LIN {X 0,Y 495.038,Z 903.66,A -85,B 0,C 180,E1 20472.506,E2 20472.506} C_VEL
LIN {X 0,Y 497.453,Z 905.615,A -85,B 0,C 180,E1 20472.244,E2 20472.244} C_VEL
LIN {X 0,Y 483.412,Z 928.293,A -85,B 0,C 180,E1 20471.672,E2 20471.672} C_VEL
LIN {X 0,Y 473.515,Z 947.117,A -85,B 0,C 180,E1 20471.077,E2 20471.077} C_VEL
LIN {X 0,Y 466.181,Z 963.721,A -85,B 0,C 180,E1 20470.451,E2 20470.451} C_VEL
LIN {X 0,Y 458.344,Z 980.789,A -85,B 0,C 180,E1 20469.812,E2 20469.812} C_VEL
LIN {X 0,Y 450.078,Z 1004.055,A -85,B 0,C 180,E1 20468.798,E2 20468.798} C_VEL
LIN {X 0,Y 447.354,Z 1025.742,A -85,B 0,C 180,E1 20468.553,E2 20468.553} C_VEL
LIN {X 0,Y 446.305,Z 1053.945,A -85,B 0,C 180,E1 20467.96,E2 20467.96} C_VEL
LIN {X 0,Y 444.603,Z 1079.758,A -85,B 0,C 180,E1 20467.185,E2 20467.185} C_VEL
LIN {X 0,Y 442.821,Z 1103.831,A -85,B 0,C 180,E1 20466.222,E2 20466.222} C_VEL
LIN {X 0,Y 440.838,Z 1127.571,A -85,B 0,C 180,E1 20465.018,E2 20465.018} C_VEL
LIN {X 0,Y 438.693,Z 1150.972,A -85,B 0,C 180,E1 20463.553,E2 20463.553} C_VEL
LIN {X 0,Y 436.639,Z 1172.47,A -85,B 0,C 180,E1 20461.936,E2 20461.936} C_VEL
LIN {X 0,Y 434.521,Z 1192.931,A -85,B 0,C 180,E1 20460.108,E2 20460.108} C_VEL
LIN {X 0,Y 432.447,Z 1212.213,A -85,B 0,C 180,E1 20458.068,E2 20458.068} C_VEL
LIN {X 0,Y 430.487,Z 1230.142,A -85,B 0,C 180,E1 20455.817,E2 20455.817} C_VEL
LIN {X 0,Y 428.709,Z 1246.625,A -85,B 0,C 180,E1 20453.359,E2 20453.359} C_VEL
LIN {X 0,Y 427.372,Z 1259.283,A -85,B 0,C 180,E1 20451.119,E2 20451.119} C_VEL
LIN {X 0,Y 426.348,Z 1269.529,A -85,B 0,C 180,E1 20449.025,E2 20449.025} C_VEL
LIN {X 0,Y 425.398,Z 1280.533,A -85,B 0,C 180,E1 20446.383,E2 20446.383} C_VEL
LIN {X 0,Y 424.715,Z 1289.348,A -85,B 0,C 180,E1 20443.756,E2 20443.756} C_VEL
LIN {X 0,Y 424.332,Z 1295.78,A -85,B 0,C 180,E1 20441.415,E2 20441.415} C_VEL
LIN {X 0,Y 424.071,Z 1301.233,A -85,B 0,C 180,E1 20438.924,E2 20438.924} C_VEL
LIN {X 0,Y 423.935,Z 1305.868,A -85,B 0,C 180,E1 20435.957,E2 20435.957} C_VEL
LIN {X 0,Y 423.908,Z 1308.176,A -85,B 0,C 180,E1 20433.516,E2 20433.516} C_VEL
LIN {X 0,Y 423.905,Z 1309.236,A -85,B 0,C 180,E1 20431.217,E2 20431.217} C_VEL
LIN {X 0,Y 423.907,Z 1309.262,A -85,B 0,C 180,E1 20428.919,E2 20428.919} C_VEL
LIN {X 0,Y 423.909,Z 1308.26,A -85,B 0,C 180,E1 20426.62,E2 20426.62} C_VEL
LIN {X 0,Y 423.937,Z 1306.164,A -85,B 0,C 180,E1 20424.316,E2 20424.316} C_VEL
LIN {X 0,Y 424.028,Z 1302.468,A -85,B 0,C 180,E1 20421.731,E2 20421.731} C_VEL
LIN {X 0,Y 424.281,Z 1296.619,A -85,B 0,C 180,E1 20418.859,E2 20418.859} C_VEL
LIN {X 0,Y 424.658,Z 1290.1,A -85,B 0,C 180,E1 20416.383,E2 20416.383} C_VEL
LIN {X 0,Y 425.229,Z 1282.608,A -85,B 0,C 180,E1 20414.032,E2 20414.032} C_VEL
LIN {X 0,Y 426.14,Z 1272.596,A -85,B 0,C 180,E1 20411.392,E2 20411.392} C_VEL
LIN {X 0,Y 427.425,Z 1260.457,A -85,B 0,C 180,E1 20408.742,E2 20408.742} C_VEL
LIN {X 0,Y 428.934,Z 1247.705,A -85,B 0,C 180,E1 20406.361,E2 20406.361} C_VEL
LIN {X 0,Y 430.988,Z 1231.433,A -85,B 0,C 180,E1 20403.773,E2 20403.773} C_VEL
LIN {X 0,Y 433.1,Z 1215.313,A -85,B 0,C 180,E1 20401.591,E2 20401.591} C_VEL
LIN {X 0,Y 435.656,Z 1196.285,A -85,B 0,C 180,E1 20399.389,E2 20399.389} C_VEL
LIN {X 0,Y 438.242,Z 1176.908,A -85,B 0,C 180,E1 20397.501,E2 20397.501} C_VEL
LIN {X 0,Y 440.756,Z 1156.929,A -85,B 0,C 180,E1 20395.852,E2 20395.852} C_VEL
LIN {X 0,Y 443.186,Z 1137.339,A -85,B 0,C 180,E1 20394.492,E2 20394.492} C_VEL
LIN {X 0,Y 445.636,Z 1115.052,A -85,B 0,C 180,E1 20393.224,E2 20393.224} C_VEL
LIN {X 0,Y 447.879,Z 1092.479,A -85,B 0,C 180,E1 20392.211,E2 20392.211} C_VEL
LIN {X 0,Y 449.738,Z 1070.105,A -85,B 0,C 180,E1 20391.457,E2 20391.457} C_VEL
LIN {X 0,Y 451.033,Z 1047.195,A -85,B 0,C 180,E1 20390.913,E2 20390.913} C_VEL
LIN {X 0,Y 452.198,Z 1021.154,A -85,B 0,C 180,E1 20390.442,E2 20390.442} C_VEL
LIN {X 0,Y 452.865,Z 1015.445,A -85,B 0,C 180,E1 20390.353,E2 20390.353} C_VEL
LIN {X 0,Y 458.36,Z 999.866,A -85,B 0,C 180,E1 20389.62,E2 20389.62} C_VEL
LIN {X 0,Y 465.063,Z 982.474,A -85,B 0,C 180,E1 20388.862,E2 20388.862} C_VEL
LIN {X 0,Y 473.981,Z 963.602,A -85,B 0,C 180,E1 20388.196,E2 20388.196} C_VEL
LIN {X 0,Y 481.845,Z 946.559,A -85,B 0,C 180,E1 20387.594,E2 20387.594} C_VEL
LIN {X 0,Y 492.91,Z 926.245,A -85,B 0,C 180,E1 20387.078,E2 20387.078} C_VEL
LIN {X 0,Y 502.453,Z 910.275,A -85,B 0,C 180,E1 20386.766,E2 20386.766} C_VEL
LIN {X 0,Y 492.063,Z 901.651,A -85,B 0,C 180,E1 20385.164,E2 20385.164} C_VEL
LIN {X 0,Y 483.388,Z 891.644,A -85,B 0,C 180,E1 20383.534,E2 20383.534} C_VEL
LIN {X 0,Y 476.69,Z 881.066,A -85,B 0,C 180,E1 20381.998,E2 20381.998} C_VEL
LIN {X 0,Y 470.917,Z 867.931,A -85,B 0,C 180,E1 20380.279,E2 20380.279} C_VEL
LIN {X 0,Y 466.996,Z 853.705,A -85,B 0,C 180,E1 20378.605,E2 20378.605} C_VEL
LIN {X 0,Y 464.773,Z 838.192,A -85,B 0,C 180,E1 20376.962,E2 20376.962} C_VEL
LIN {X 0,Y 464.211,Z 820.272,A -85,B 0,C 180,E1 20375.256,E2 20375.256} C_VEL
LIN {X 0,Y 465.72,Z 798.884,A -85,B 0,C 180,E1 20373.439,E2 20373.439} C_VEL
LIN {X 0,Y 470.117,Z 762.904,A -85,B 0,C 180,E1 20370.551,E2 20370.551} C_VEL
LIN {X 0,Y 460.348,Z 744.289,A -85,B 0,C 180,E1 20367.136,E2 20367.136} C_VEL
LIN {X 0,Y 452.253,Z 729.507,A -85,B 0,C 180,E1 20364.142,E2 20364.142} C_VEL
LIN {X 0,Y 444.794,Z 716.18,A -85,B 0,C 180,E1 20361.217,E2 20361.217} C_VEL
LIN {X 0,Y 439.088,Z 706.262,A -85,B 0,C 180,E1 20358.865,E2 20358.865} C_VEL
LIN {X 0,Y 436.138,Z 701.205,A -85,B 0,C 180,E1 20357.614,E2 20357.614} C_VEL
LIN {X 0,Y 433.616,Z 696.697,A -85,B 0,C 180,E1 20356.476,E2 20356.476} C_VEL
LIN {X 0,Y 431.403,Z 692.701,A -85,B 0,C 180,E1 20355.458,E2 20355.458} C_VEL
LIN {X 0,Y 428.801,Z 688.643,A -85,B 0,C 180,E1 20354.31,E2 20354.31} C_VEL
LIN {X 0,Y 428.14,Z 686.924,A -85,B 0,C 180,E1 20353.918,E2 20353.918} C_VEL
LIN {X 0,Y 425.994,Z 684.148,A -85,B 0,C 180,E1 20353.022,E2 20353.022} C_VEL
LIN {X 0,Y 425.314,Z 681.755,A -85,B 0,C 180,E1 20352.49,E2 20352.49} C_VEL
LIN {X 0,Y 425.312,Z 681.753,A -85,B 0,C 180,E1 20348.653,E2 20348.653} C_VEL
LIN {X 0,Y 425.318,Z 681.753,A -85,B 0,C 180,E1 20344.854,E2 20344.854} C_VEL
LIN {X 0,Y 425.322,Z 681.753,A -85,B 0,C 180,E1 20340.943,E2 20340.943} C_VEL
LIN {X 0,Y 425.312,Z 681.758,A -85,B 0,C 180,E1 20337.035,E2 20337.035} C_VEL
LIN {X 0,Y 425.322,Z 681.755,A -85,B 0,C 180,E1 20333.249,E2 20333.249} C_VEL
LIN {X 0,Y 425.313,Z 681.754,A -85,B 0,C 180,E1 20329.297,E2 20329.297} C_VEL
LIN {X 0,Y 425.324,Z 681.757,A -85,B 0,C 180,E1 20325.431,E2 20325.431} C_VEL
LIN {X 0,Y 425.307,Z 681.749,A -85,B 0,C 180,E1 20321.638,E2 20321.638} C_VEL
LIN {X 0,Y 425.321,Z 681.751,A -85,B 0,C 180,E1 20317.852,E2 20317.852} C_VEL
LIN {X 0,Y 425.311,Z 681.752,A -85,B 0,C 180,E1 20313.92,E2 20313.92} C_VEL
LIN {X 0,Y 425.309,Z 681.71,A -85,B 0,C 180,E1 20310.106,E2 20310.106} C_VEL
LIN {X 0,Y 425.31,Z 681.734,A -85,B 0,C 180,E1 20306.302,E2 20306.302} C_VEL
LIN {X 0,Y 425.319,Z 681.749,A -85,B 0,C 180,E1 20302.393,E2 20302.393} C_VEL
LIN {X 0,Y 425.341,Z 681.936,A -85,B 0,C 180,E1 20299.775,E2 20299.775} C_VEL
LIN {X 0,Y 426.485,Z 685.003,A -85,B 0,C 180,E1 20299.326,E2 20299.326} C_VEL
LIN {X 0,Y 427.836,Z 686.906,A -85,B 0,C 180,E1 20298.951,E2 20298.951} C_VEL
LIN {X 0,Y 436.635,Z 704.262,A -85,B 0,C 180,E1 20296.163,E2 20296.163} C_VEL
LIN {X 0,Y 444.835,Z 722.235,A -85,B 0,C 180,E1 20293.54,E2 20293.54} C_VEL
LIN {X 0,Y 451.168,Z 737.937,A -85,B 0,C 180,E1 20291.462,E2 20291.462} C_VEL
LIN {X 0,Y 449.321,Z 772.77,A -85,B 0,C 180,E1 20288.908,E2 20288.908} C_VEL
LIN {X 0,Y 452.478,Z 796.072,A -85,B 0,C 180,E1 20288.098,E2 20288.098} C_VEL
LIN {X 0,Y 447.843,Z 982.654,A -85,B 0,C 180,E1 20284.884,E2 20284.884} C_VEL
LIN {X 0,Y 446.814,Z 990.345,A -85,B 0,C 180,E1 20284.828,E2 20284.828} C_VEL
LIN {X 0,Y 441.207,Z 1010.823,A -85,B 0,C 180,E1 20284.942,E2 20284.942} C_VEL
LIN {X 0,Y 440.46,Z 1017.42,A -85,B 0,C 180,E1 20284.882,E2 20284.882} C_VEL
LIN {X 0,Y 439.652,Z 1041.722,A -85,B 0,C 180,E1 20284.384,E2 20284.384} C_VEL
LIN {X 0,Y 438.49,Z 1062.151,A -85,B 0,C 180,E1 20283.731,E2 20283.731} C_VEL
LIN {X 0,Y 436.883,Z 1082.14,A -85,B 0,C 180,E1 20282.846,E2 20282.846} C_VEL
LIN {X 0,Y 434.833,Z 1101.923,A -85,B 0,C 180,E1 20281.703,E2 20281.703} C_VEL
LIN {X 0,Y 432.657,Z 1119.868,A -85,B 0,C 180,E1 20280.404,E2 20280.404} C_VEL
LIN {X 0,Y 430.326,Z 1137,A -85,B 0,C 180,E1 20278.899,E2 20278.899} C_VEL
LIN {X 0,Y 427.83,Z 1153.912,A -85,B 0,C 180,E1 20277.111,E2 20277.111} C_VEL
LIN {X 0,Y 425.441,Z 1169.228,A -85,B 0,C 180,E1 20275.174,E2 20275.174} C_VEL
LIN {X 0,Y 423.25,Z 1183.135,A -85,B 0,C 180,E1 20273.087,E2 20273.087} C_VEL
LIN {X 0,Y 421.188,Z 1196.357,A -85,B 0,C 180,E1 20270.714,E2 20270.714} C_VEL
LIN {X 0,Y 419.467,Z 1207.988,A -85,B 0,C 180,E1 20268.195,E2 20268.195} C_VEL
LIN {X 0,Y 418.183,Z 1217.584,A -85,B 0,C 180,E1 20265.674,E2 20265.674} C_VEL
LIN {X 0,Y 417.232,Z 1225.83,A -85,B 0,C 180,E1 20263.018,E2 20263.018} C_VEL
LIN {X 0,Y 416.614,Z 1232.642,A -85,B 0,C 180,E1 20260.229,E2 20260.229} C_VEL
LIN {X 0,Y 416.268,Z 1237.71,A -85,B 0,C 180,E1 20257.452,E2 20257.452} C_VEL
LIN {X 0,Y 416.123,Z 1241.146,A -85,B 0,C 180,E1 20254.685,E2 20254.685} C_VEL
LIN {X 0,Y 416.061,Z 1242.953,A -85,B 0,C 180,E1 20251.927,E2 20251.927} C_VEL
LIN {X 0,Y 416.051,Z 1243.266,A -85,B 0,C 180,E1 20249.173,E2 20249.173} C_VEL
LIN {X 0,Y 416.084,Z 1241.986,A -85,B 0,C 180,E1 20246.279,E2 20246.279} C_VEL
LIN {X 0,Y 416.201,Z 1239.212,A -85,B 0,C 180,E1 20243.516,E2 20243.516} C_VEL
LIN {X 0,Y 416.476,Z 1234.648,A -85,B 0,C 180,E1 20240.651,E2 20240.651} C_VEL
LIN {X 0,Y 417.001,Z 1228.327,A -85,B 0,C 180,E1 20237.818,E2 20237.818} C_VEL
LIN {X 0,Y 417.812,Z 1220.676,A -85,B 0,C 180,E1 20235.163,E2 20235.163} C_VEL
LIN {X 0,Y 419.021,Z 1211.164,A -85,B 0,C 180,E1 20232.502,E2 20232.502} C_VEL
LIN {X 0,Y 420.599,Z 1200.172,A -85,B 0,C 180,E1 20229.981,E2 20229.981} C_VEL
LIN {X 0,Y 422.519,Z 1187.715,A -85,B 0,C 180,E1 20227.604,E2 20227.604} C_VEL
LIN {X 0,Y 424.661,Z 1174.241,A -85,B 0,C 180,E1 20225.444,E2 20225.444} C_VEL
LIN {X 0,Y 427.02,Z 1159.32,A -85,B 0,C 180,E1 20223.434,E2 20223.434} C_VEL
LIN {X 0,Y 429.529,Z 1142.738,A -85,B 0,C 180,E1 20221.573,E2 20221.573} C_VEL
LIN {X 0,Y 431.905,Z 1125.625,A -85,B 0,C 180,E1 20219.976,E2 20219.976} C_VEL
LIN {X 0,Y 434.113,Z 1108.191,A -85,B 0,C 180,E1 20218.632,E2 20218.632} C_VEL
LIN {X 0,Y 436.16,Z 1089.5,A -85,B 0,C 180,E1 20217.458,E2 20217.458} C_VEL
LIN {X 0,Y 437.911,Z 1069.932,A -85,B 0,C 180,E1 20216.492,E2 20216.492} C_VEL
LIN {X 0,Y 439.299,Z 1049.695,A -85,B 0,C 180,E1 20215.747,E2 20215.747} C_VEL
LIN {X 0,Y 440.181,Z 1028.656,A -85,B 0,C 180,E1 20215.225,E2 20215.225} C_VEL
LIN {X 0,Y 445.986,Z 805.37,A -85,B 0,C 180,E1 20211.329,E2 20211.329} C_VEL
LIN {X 0,Y 439.438,Z 775.543,A -85,B 0,C 180,E1 20209.995,E2 20209.995} C_VEL
LIN {X 0,Y 440.967,Z 748.497,A -85,B 0,C 180,E1 20207.138,E2 20207.138} C_VEL
LIN {X 0,Y 441.382,Z 741.584,A -85,B 0,C 180,E1 20206.366,E2 20206.366} C_VEL
LIN {X 0,Y 435.004,Z 723.036,A -85,B 0,C 180,E1 20203.228,E2 20203.228} C_VEL
LIN {X 0,Y 432.196,Z 715.931,A -85,B 0,C 180,E1 20201.896,E2 20201.896} C_VEL
LIN {X 0,Y 439.21,Z 733.497,A -85,B 0,C 180,E1 20198.974,E2 20198.974} C_VEL
LIN {X 0,Y 441.605,Z 740.146,A -85,B 0,C 180,E1 20197.94,E2 20197.94} C_VEL
LIN {X 0,Y 437.922,Z 777.868,A -85,B 0,C 180,E1 20194.171,E2 20194.171} C_VEL
LIN {X 0,Y 434.268,Z 818.23,A -85,B 0,C 180,E1 20190.204,E2 20190.204} C_VEL
LIN {X 0,Y 430.923,Z 859.713,A -85,B 0,C 180,E1 20186.195,E2 20186.195} C_VEL
LIN {X 0,Y 432.214,Z 869.718,A -85,B 0,C 180,E1 20185.864,E2 20185.864} C_VEL
LIN {X 0,Y 427.104,Z 1030.884,A -85,B 0,C 180,E1 20182.45,E2 20182.45} C_VEL
LIN {X 0,Y 426.473,Z 1049.018,A -85,B 0,C 180,E1 20181.798,E2 20181.798} C_VEL
LIN {X 0,Y 425.572,Z 1066.146,A -85,B 0,C 180,E1 20180.923,E2 20180.923} C_VEL
LIN {X 0,Y 424.468,Z 1082.264,A -85,B 0,C 180,E1 20179.828,E2 20179.828} C_VEL
LIN {X 0,Y 423.182,Z 1098.056,A -85,B 0,C 180,E1 20178.458,E2 20178.458} C_VEL
LIN {X 0,Y 421.941,Z 1112.066,A -85,B 0,C 180,E1 20176.946,E2 20176.946} C_VEL
LIN {X 0,Y 420.715,Z 1124.974,A -85,B 0,C 180,E1 20175.227,E2 20175.227} C_VEL
LIN {X 0,Y 419.625,Z 1136.357,A -85,B 0,C 180,E1 20173.364,E2 20173.364} C_VEL
LIN {X 0,Y 418.669,Z 1146.634,A -85,B 0,C 180,E1 20171.294,E2 20171.294} C_VEL
LIN {X 0,Y 417.983,Z 1154.845,A -85,B 0,C 180,E1 20169.223,E2 20169.223} C_VEL
LIN {X 0,Y 417.505,Z 1161.626,A -85,B 0,C 180,E1 20167.016,E2 20167.016} C_VEL
LIN {X 0,Y 417.185,Z 1166.965,A -85,B 0,C 180,E1 20164.674,E2 20164.674} C_VEL
LIN {X 0,Y 417.06,Z 1170.567,A -85,B 0,C 180,E1 20162.336,E2 20162.336} C_VEL
LIN {X 0,Y 417.033,Z 1172.511,A -85,B 0,C 180,E1 20160,E2 20160} C_VEL
LIN {X 0,Y 417.114,Z 1172.754,A -85,B 0,C 180,E1 20157.527,E2 20157.527} C_VEL
LIN {X 0,Y 417.305,Z 1171.255,A -85,B 0,C 180,E1 20155.052,E2 20155.052} C_VEL
LIN {X 0,Y 417.655,Z 1168.127,A -85,B 0,C 180,E1 20152.711,E2 20152.711} C_VEL
LIN {X 0,Y 418.17,Z 1163.204,A -85,B 0,C 180,E1 20150.365,E2 20150.365} C_VEL
LIN {X 0,Y 418.907,Z 1156.744,A -85,B 0,C 180,E1 20148.127,E2 20148.127} C_VEL
LIN {X 0,Y 419.852,Z 1149.051,A -85,B 0,C 180,E1 20146.083,E2 20146.083} C_VEL
LIN {X 0,Y 421.073,Z 1139.143,A -85,B 0,C 180,E1 20144.012,E2 20144.012} C_VEL
LIN {X 0,Y 422.333,Z 1128.513,A -85,B 0,C 180,E1 20142.218,E2 20142.218} C_VEL
LIN {X 0,Y 423.684,Z 1116.426,A -85,B 0,C 180,E1 20140.565,E2 20140.565} C_VEL
LIN {X 0,Y 424.997,Z 1103.344,A -85,B 0,C 180,E1 20139.12,E2 20139.12} C_VEL
LIN {X 0,Y 426.261,Z 1088.579,A -85,B 0,C 180,E1 20137.812,E2 20137.812} C_VEL
LIN {X 0,Y 427.235,Z 1073.625,A -85,B 0,C 180,E1 20136.776,E2 20136.776} C_VEL
LIN {X 0,Y 427.984,Z 1057.21,A -85,B 0,C 180,E1 20135.924,E2 20135.924} C_VEL
LIN {X 0,Y 428.393,Z 1040.561,A -85,B 0,C 180,E1 20135.32,E2 20135.32} C_VEL
LIN {X 0,Y 430.053,Z 1004.28,A -85,B 0,C 180,E1 20134.281,E2 20134.281} C_VEL
LIN {X 0,Y 435.783,Z 934.51,A -85,B 0,C 180,E1 20132.18,E2 20132.18} C_VEL
LIN {X 0,Y 439.664,Z 897.058,A -85,B 0,C 180,E1 20131.028,E2 20131.028} C_VEL
LIN {X 0,Y 448.187,Z 879.223,A -85,B 0,C 180,E1 20129.723,E2 20129.723} C_VEL
LIN {X 0,Y 455.611,Z 858.642,A -85,B 0,C 180,E1 20127.027,E2 20127.027} C_VEL
LIN {X 0,Y 463.426,Z 843.098,A -85,B 0,C 180,E1 20124.826,E2 20124.826} C_VEL
LIN {X 0,Y 466.032,Z 838.935,A -85,B 0,C 180,E1 20124.169,E2 20124.169} C_VEL
LIN {X 0,Y 461.288,Z 847.431,A -85,B 0,C 180,E1 20122.634,E2 20122.634} C_VEL
LIN {X 0,Y 458.913,Z 855.669,A -85,B 0,C 180,E1 20121.136,E2 20121.136} C_VEL
LIN {X 0,Y 458.654,Z 864.038,A -85,B 0,C 180,E1 20119.65,E2 20119.65} C_VEL
LIN {X 0,Y 460.551,Z 872.948,A -85,B 0,C 180,E1 20118.13,E2 20118.13} C_VEL
LIN {X 0,Y 464.57,Z 882.06,A -85,B 0,C 180,E1 20116.642,E2 20116.642} C_VEL
LIN {X 0,Y 471.408,Z 892.115,A -85,B 0,C 180,E1 20115.066,E2 20115.066} C_VEL
LIN {X 0,Y 480.465,Z 901.866,A -85,B 0,C 180,E1 20113.598,E2 20113.598} C_VEL
LIN {X 0,Y 487.937,Z 908.356,A -85,B 0,C 180,E1 20112.653,E2 20112.653} C_VEL
LIN {X 0,Y 474.992,Z 929.987,A -85,B 0,C 180,E1 20112.102,E2 20112.102} C_VEL
LIN {X 0,Y 465.553,Z 948.61,A -85,B 0,C 180,E1 20111.496,E2 20111.496} C_VEL
LIN {X 0,Y 459.591,Z 962.152,A -85,B 0,C 180,E1 20110.983,E2 20110.983} C_VEL
LIN {X 0,Y 451.744,Z 979.218,A -85,B 0,C 180,E1 20110.346,E2 20110.346} C_VEL
LIN {X 0,Y 443.804,Z 1001.344,A -85,B 0,C 180,E1 20109.392,E2 20109.392} C_VEL
LIN {X 0,Y 440.661,Z 1025.004,A -85,B 0,C 180,E1 20109.121,E2 20109.121} C_VEL
LIN {X 0,Y 439.441,Z 1052.21,A -85,B 0,C 180,E1 20108.517,E2 20108.517} C_VEL
LIN {X 0,Y 437.473,Z 1079.547,A -85,B 0,C 180,E1 20107.664,E2 20107.664} C_VEL
LIN {X 0,Y 435.503,Z 1103.803,A -85,B 0,C 180,E1 20106.651,E2 20106.651} C_VEL
LIN {X 0,Y 433.346,Z 1127.664,A -85,B 0,C 180,E1 20105.39,E2 20105.39} C_VEL
LIN {X 0,Y 431.111,Z 1150.734,A -85,B 0,C 180,E1 20103.903,E2 20103.903} C_VEL
LIN {X 0,Y 428.965,Z 1171.999,A -85,B 0,C 180,E1 20102.261,E2 20102.261} C_VEL
LIN {X 0,Y 426.717,Z 1192.757,A -85,B 0,C 180,E1 20100.353,E2 20100.353} C_VEL
LIN {X 0,Y 424.623,Z 1211.534,A -85,B 0,C 180,E1 20098.318,E2 20098.318} C_VEL
LIN {X 0,Y 422.618,Z 1229.421,A -85,B 0,C 180,E1 20096.032,E2 20096.032} C_VEL
LIN {X 0,Y 420.881,Z 1245.063,A -85,B 0,C 180,E1 20093.671,E2 20093.671} C_VEL
LIN {X 0,Y 419.424,Z 1258.641,A -85,B 0,C 180,E1 20091.237,E2 20091.237} C_VEL
LIN {X 0,Y 418.253,Z 1270.243,A -85,B 0,C 180,E1 20088.799,E2 20088.799} C_VEL
LIN {X 0,Y 417.339,Z 1280.823,A -85,B 0,C 180,E1 20086.115,E2 20086.115} C_VEL
LIN {X 0,Y 416.722,Z 1288.995,A -85,B 0,C 180,E1 20083.6,E2 20083.6} C_VEL
LIN {X 0,Y 416.321,Z 1295.999,A -85,B 0,C 180,E1 20080.938,E2 20080.938} C_VEL
LIN {X 0,Y 416.096,Z 1301.766,A -85,B 0,C 180,E1 20078.012,E2 20078.012} C_VEL
LIN {X 0,Y 416.013,Z 1305.223,A -85,B 0,C 180,E1 20075.517,E2 20075.517} C_VEL
LIN {X 0,Y 415.98,Z 1307.397,A -85,B 0,C 180,E1 20073.032,E2 20073.032} C_VEL
LIN {X 0,Y 415.966,Z 1308.359,A -85,B 0,C 180,E1 20070.414,E2 20070.414} C_VEL
LIN {X 0,Y 415.969,Z 1307.708,A -85,B 0,C 180,E1 20067.383,E2 20067.383} C_VEL
LIN {X 0,Y 415.991,Z 1305.624,A -85,B 0,C 180,E1 20064.76,E2 20064.76} C_VEL
LIN {X 0,Y 416.052,Z 1302.577,A -85,B 0,C 180,E1 20062.405,E2 20062.405} C_VEL
LIN {X 0,Y 416.213,Z 1298.127,A -85,B 0,C 180,E1 20059.901,E2 20059.901} C_VEL
LIN {X 0,Y 416.575,Z 1291.255,A -85,B 0,C 180,E1 20056.961,E2 20056.961} C_VEL
LIN {X 0,Y 417.196,Z 1282.731,A -85,B 0,C 180,E1 20054.145,E2 20054.145} C_VEL
LIN {X 0,Y 418.054,Z 1273.461,A -85,B 0,C 180,E1 20051.597,E2 20051.597} C_VEL
LIN {X 0,Y 419.398,Z 1261.083,A -85,B 0,C 180,E1 20048.755,E2 20048.755} C_VEL
LIN {X 0,Y 421.026,Z 1247.771,A -85,B 0,C 180,E1 20046.19,E2 20046.19} C_VEL
LIN {X 0,Y 423.131,Z 1231.902,A -85,B 0,C 180,E1 20043.582,E2 20043.582} C_VEL
LIN {X 0,Y 425.572,Z 1214.202,A -85,B 0,C 180,E1 20041.132,E2 20041.132} C_VEL
LIN {X 0,Y 428.213,Z 1195.527,A -85,B 0,C 180,E1 20038.935,E2 20038.935} C_VEL
LIN {X 0,Y 430.898,Z 1176.361,A -85,B 0,C 180,E1 20037.035,E2 20037.035} C_VEL
LIN {X 0,Y 433.683,Z 1155.522,A -85,B 0,C 180,E1 20035.288,E2 20035.288} C_VEL
LIN {X 0,Y 436.236,Z 1135.896,A -85,B 0,C 180,E1 20033.911,E2 20033.911} C_VEL
LIN {X 0,Y 438.86,Z 1113.272,A -85,B 0,C 180,E1 20032.616,E2 20032.616} C_VEL
LIN {X 0,Y 441.186,Z 1091.062,A -85,B 0,C 180,E1 20031.614,E2 20031.614} C_VEL
LIN {X 0,Y 443.127,Z 1068.649,A -85,B 0,C 180,E1 20030.854,E2 20030.854} C_VEL
LIN {X 0,Y 444.492,Z 1045.664,A -85,B 0,C 180,E1 20030.301,E2 20030.301} C_VEL
LIN {X 0,Y 445.693,Z 1021.042,A -85,B 0,C 180,E1 20029.848,E2 20029.848} C_VEL
LIN {X 0,Y 446.436,Z 1014.488,A -85,B 0,C 180,E1 20029.75,E2 20029.75} C_VEL
LIN {X 0,Y 455.582,Z 989.278,A -85,B 0,C 180,E1 20028.572,E2 20028.572} C_VEL
LIN {X 0,Y 462.727,Z 973.075,A -85,B 0,C 180,E1 20027.946,E2 20027.946} C_VEL
LIN {X 0,Y 467.756,Z 962.742,A -85,B 0,C 180,E1 20027.593,E2 20027.593} C_VEL
LIN {X 0,Y 475.644,Z 945.671,A -85,B 0,C 180,E1 20026.99,E2 20026.99} C_VEL
LIN {X 0,Y 486.388,Z 925.992,A -85,B 0,C 180,E1 20026.477,E2 20026.477} C_VEL
LIN {X 0,Y 493.613,Z 913.634,A -85,B 0,C 180,E1 20026.219,E2 20026.219} C_VEL
LIN {X 0,Y 483.977,Z 904.743,A -85,B 0,C 180,E1 20024.621,E2 20024.621} C_VEL
LIN {X 0,Y 475.042,Z 893.384,A -85,B 0,C 180,E1 20022.831,E2 20022.831} C_VEL
LIN {X 0,Y 468.188,Z 880.931,A -85,B 0,C 180,E1 20021.075,E2 20021.075} C_VEL
LIN {X 0,Y 463.09,Z 867.139,A -85,B 0,C 180,E1 20019.323,E2 20019.323} C_VEL
LIN {X 0,Y 459.657,Z 851.33,A -85,B 0,C 180,E1 20017.521,E2 20017.521} C_VEL
LIN {X 0,Y 458.099,Z 833.67,A -85,B 0,C 180,E1 20015.716,E2 20015.716} C_VEL
LIN {X 0,Y 458.454,Z 815.294,A -85,B 0,C 180,E1 20014.03,E2 20014.03} C_VEL
LIN {X 0,Y 461.9,Z 784.161,A -85,B 0,C 180,E1 20011.475,E2 20011.475} C_VEL
LIN {X 0,Y 463.978,Z 767.026,A -85,B 0,C 180,E1 20010.068,E2 20010.068} C_VEL
LIN {X 0,Y 454.764,Z 749.481,A -85,B 0,C 180,E1 20006.789,E2 20006.789} C_VEL
LIN {X 0,Y 446.694,Z 734.635,A -85,B 0,C 180,E1 20003.759,E2 20003.759} C_VEL
LIN {X 0,Y 439.258,Z 721.343,A -85,B 0,C 180,E1 20000.799,E2 20000.799} C_VEL
LIN {X 0,Y 434.17,Z 712.393,A -85,B 0,C 180,E1 19998.669,E2 19998.669} C_VEL
LIN {X 0,Y 428.67,Z 702.79,A -85,B 0,C 180,E1 19996.254,E2 19996.254} C_VEL
LIN {X 0,Y 425.558,Z 697.521,A -85,B 0,C 180,E1 19994.838,E2 19994.838} C_VEL
LIN {X 0,Y 422.818,Z 692.726,A -85,B 0,C 180,E1 19993.539,E2 19993.539} C_VEL
LIN {X 0,Y 420.639,Z 689.033,A -85,B 0,C 180,E1 19992.492,E2 19992.492} C_VEL
LIN {X 0,Y 419.862,Z 687.604,A -85,B 0,C 180,E1 19992.096,E2 19992.096} C_VEL
LIN {X 0,Y 417.877,Z 684.695,A -85,B 0,C 180,E1 19991.175,E2 19991.175} C_VEL
LIN {X 0,Y 417.377,Z 682.743,A -85,B 0,C 180,E1 19990.699,E2 19990.699} C_VEL
LIN {X 0,Y 417.379,Z 682.742,A -85,B 0,C 180,E1 19986.879,E2 19986.879} C_VEL
LIN {X 0,Y 417.371,Z 682.744,A -85,B 0,C 180,E1 19983.021,E2 19983.021} C_VEL
LIN {X 0,Y 417.373,Z 682.746,A -85,B 0,C 180,E1 19979.176,E2 19979.176} C_VEL
LIN {X 0,Y 417.378,Z 682.745,A -85,B 0,C 180,E1 19975.233,E2 19975.233} C_VEL
LIN {X 0,Y 417.369,Z 682.742,A -85,B 0,C 180,E1 19971.458,E2 19971.458} C_VEL
LIN {X 0,Y 417.383,Z 682.746,A -85,B 0,C 180,E1 19967.549,E2 19967.549} C_VEL
LIN {X 0,Y 417.378,Z 682.744,A -85,B 0,C 180,E1 19963.723,E2 19963.723} C_VEL
LIN {X 0,Y 417.38,Z 682.738,A -85,B 0,C 180,E1 19959.674,E2 19959.674} C_VEL
LIN {X 0,Y 417.376,Z 682.738,A -85,B 0,C 180,E1 19955.817,E2 19955.817} C_VEL
LIN {X 0,Y 417.381,Z 682.691,A -85,B 0,C 180,E1 19951.84,E2 19951.84} C_VEL
LIN {X 0,Y 417.377,Z 682.747,A -85,B 0,C 180,E1 19947.871,E2 19947.871} C_VEL
LIN {X 0,Y 417.374,Z 682.699,A -85,B 0,C 180,E1 19944.061,E2 19944.061} C_VEL
LIN {X 0,Y 417.409,Z 682.942,A -85,B 0,C 180,E1 19940.904,E2 19940.904} C_VEL
LIN {X 0,Y 418.703,Z 686.241,A -85,B 0,C 180,E1 19940.387,E2 19940.387} C_VEL
LIN {X 0,Y 420.031,Z 688.111,A -85,B 0,C 180,E1 19940.005,E2 19940.005} C_VEL
LIN {X 0,Y 427.309,Z 702.116,A -85,B 0,C 180,E1 19937.632,E2 19937.632} C_VEL
LIN {X 0,Y 435.07,Z 718.261,A -85,B 0,C 180,E1 19935.127,E2 19935.127} C_VEL
LIN {X 0,Y 442.718,Z 736.348,A -85,B 0,C 180,E1 19932.586,E2 19932.586} C_VEL
LIN {X 0,Y 444.713,Z 741.787,A -85,B 0,C 180,E1 19931.893,E2 19931.893} C_VEL
LIN {X 0,Y 442.988,Z 773.784,A -85,B 0,C 180,E1 19929.543,E2 19929.543} C_VEL
LIN {X 0,Y 446.195,Z 797.463,A -85,B 0,C 180,E1 19928.714,E2 19928.714} C_VEL
LIN {X 0,Y 440.46,Z 1017.42,A -85,B 0,C 180,E1 19924.882,E2 19924.882} C_VEL
LIN {X 0,Y 439.481,Z 1025.113,A -85,B 0,C 180,E1 19924.821,E2 19924.821} C_VEL
LIN {X 0,Y 433.861,Z 1044.431,A -85,B 0,C 180,E1 19924.852,E2 19924.852} C_VEL
LIN {X 0,Y 432.59,Z 1051.974,A -85,B 0,C 180,E1 19924.697,E2 19924.697} C_VEL
LIN {X 0,Y 431.112,Z 1072.393,A -85,B 0,C 180,E1 19923.92,E2 19923.92} C_VEL
LIN {X 0,Y 429.169,Z 1092.68,A -85,B 0,C 180,E1 19922.876,E2 19922.876} C_VEL
LIN {X 0,Y 427.063,Z 1110.528,A -85,B 0,C 180,E1 19921.708,E2 19921.708} C_VEL
LIN {X 0,Y 424.612,Z 1128.636,A -85,B 0,C 180,E1 19920.259,E2 19920.259} C_VEL
LIN {X 0,Y 421.957,Z 1146.438,A -85,B 0,C 180,E1 19918.519,E2 19918.519} C_VEL
LIN {X 0,Y 419.337,Z 1162.711,A -85,B 0,C 180,E1 19916.601,E2 19916.601} C_VEL
LIN {X 0,Y 417.02,Z 1176.626,A -85,B 0,C 180,E1 19914.656,E2 19914.656} C_VEL
LIN {X 0,Y 414.74,Z 1190.269,A -85,B 0,C 180,E1 19912.389,E2 19912.389} C_VEL
LIN {X 0,Y 412.753,Z 1202.417,A -85,B 0,C 180,E1 19909.965,E2 19909.965} C_VEL
LIN {X 0,Y 411.121,Z 1213.084,A -85,B 0,C 180,E1 19907.405,E2 19907.405} C_VEL
LIN {X 0,Y 409.876,Z 1222.33,A -85,B 0,C 180,E1 19904.696,E2 19904.696} C_VEL
LIN {X 0,Y 409.001,Z 1230.077,A -85,B 0,C 180,E1 19901.849,E2 19901.849} C_VEL
LIN {X 0,Y 408.483,Z 1235.998,A -85,B 0,C 180,E1 19899.012,E2 19899.012} C_VEL
LIN {X 0,Y 408.22,Z 1240.242,A -85,B 0,C 180,E1 19896.186,E2 19896.186} C_VEL
LIN {X 0,Y 408.108,Z 1242.849,A -85,B 0,C 180,E1 19893.37,E2 19893.37} C_VEL
LIN {X 0,Y 408.073,Z 1243.904,A -85,B 0,C 180,E1 19890.561,E2 19890.561} C_VEL
LIN {X 0,Y 408.089,Z 1243.41,A -85,B 0,C 180,E1 19887.612,E2 19887.612} C_VEL
LIN {X 0,Y 408.161,Z 1241.401,A -85,B 0,C 180,E1 19884.799,E2 19884.799} C_VEL
LIN {X 0,Y 408.366,Z 1237.843,A -85,B 0,C 180,E1 19881.977,E2 19881.977} C_VEL
LIN {X 0,Y 408.793,Z 1232.28,A -85,B 0,C 180,E1 19879.001,E2 19879.001} C_VEL
LIN {X 0,Y 409.539,Z 1225.137,A -85,B 0,C 180,E1 19876.157,E2 19876.157} C_VEL
LIN {X 0,Y 410.637,Z 1216.534,A -85,B 0,C 180,E1 19873.448,E2 19873.448} C_VEL
LIN {X 0,Y 412.101,Z 1206.537,A -85,B 0,C 180,E1 19870.88,E2 19870.88} C_VEL
LIN {X 0,Y 414.028,Z 1194.457,A -85,B 0,C 180,E1 19868.315,E2 19868.315} C_VEL
LIN {X 0,Y 416.181,Z 1181.642,A -85,B 0,C 180,E1 19866.045,E2 19866.045} C_VEL
LIN {X 0,Y 418.588,Z 1167.352,A -85,B 0,C 180,E1 19863.914,E2 19863.914} C_VEL
LIN {X 0,Y 421.267,Z 1151.035,A -85,B 0,C 180,E1 19861.885,E2 19861.885} C_VEL
LIN {X 0,Y 423.968,Z 1133.464,A -85,B 0,C 180,E1 19860.08,E2 19860.08} C_VEL
LIN {X 0,Y 426.449,Z 1115.483,A -85,B 0,C 180,E1 19858.563,E2 19858.563} C_VEL
LIN {X 0,Y 428.643,Z 1097.357,A -85,B 0,C 180,E1 19857.316,E2 19857.316} C_VEL
LIN {X 0,Y 430.627,Z 1077.904,A -85,B 0,C 180,E1 19856.25,E2 19856.25} C_VEL
LIN {X 0,Y 432.213,Z 1057.603,A -85,B 0,C 180,E1 19855.402,E2 19855.402} C_VEL
LIN {X 0,Y 433.344,Z 1037.279,A -85,B 0,C 180,E1 19854.802,E2 19854.802} C_VEL
LIN {X 0,Y 434.933,Z 980.927,A -85,B 0,C 180,E1 19853.772,E2 19853.772} C_VEL
LIN {X 0,Y 439.656,Z 806.629,A -85,B 0,C 180,E1 19850.683,E2 19850.683} C_VEL
LIN {X 0,Y 433.025,Z 776.132,A -85,B 0,C 180,E1 19849.283,E2 19849.283} C_VEL
LIN {X 0,Y 434.656,Z 748.706,A -85,B 0,C 180,E1 19846.361,E2 19846.361} C_VEL
LIN {X 0,Y 434.756,Z 745.153,A -85,B 0,C 180,E1 19845.957,E2 19845.957} C_VEL
LIN {X 0,Y 429.003,Z 728.262,A -85,B 0,C 180,E1 19843.07,E2 19843.07} C_VEL
LIN {X 0,Y 426.593,Z 722.044,A -85,B 0,C 180,E1 19841.889,E2 19841.889} C_VEL
LIN {X 0,Y 433.637,Z 740.063,A -85,B 0,C 180,E1 19838.894,E2 19838.894} C_VEL
LIN {X 0,Y 434.863,Z 743.959,A -85,B 0,C 180,E1 19838.299,E2 19838.299} C_VEL
LIN {X 0,Y 430.976,Z 781.828,A -85,B 0,C 180,E1 19834.477,E2 19834.477} C_VEL
LIN {X 0,Y 427.091,Z 823.195,A -85,B 0,C 180,E1 19830.377,E2 19830.377} C_VEL
LIN {X 0,Y 423.997,Z 861.201,A -85,B 0,C 180,E1 19826.698,E2 19826.698} C_VEL
LIN {X 0,Y 425.2,Z 870.846,A -85,B 0,C 180,E1 19826.366,E2 19826.366} C_VEL
LIN {X 0,Y 419.728,Z 1032.193,A -85,B 0,C 180,E1 19822.849,E2 19822.849} C_VEL
LIN {X 0,Y 419.06,Z 1050.35,A -85,B 0,C 180,E1 19822.177,E2 19822.177} C_VEL
LIN {X 0,Y 418.148,Z 1066.952,A -85,B 0,C 180,E1 19821.313,E2 19821.313} C_VEL
LIN {X 0,Y 416.998,Z 1083.155,A -85,B 0,C 180,E1 19820.199,E2 19820.199} C_VEL
LIN {X 0,Y 415.715,Z 1098.272,A -85,B 0,C 180,E1 19818.875,E2 19818.875} C_VEL
LIN {X 0,Y 414.404,Z 1112.447,A -85,B 0,C 180,E1 19817.336,E2 19817.336} C_VEL
LIN {X 0,Y 413.108,Z 1125.571,A -85,B 0,C 180,E1 19815.585,E2 19815.585} C_VEL
LIN {X 0,Y 411.911,Z 1137.449,A -85,B 0,C 180,E1 19813.619,E2 19813.619} C_VEL
LIN {X 0,Y 410.899,Z 1147.773,A -85,B 0,C 180,E1 19811.51,E2 19811.51} C_VEL
LIN {X 0,Y 410.168,Z 1156.038,A -85,B 0,C 180,E1 19809.4,E2 19809.4} C_VEL
LIN {X 0,Y 409.656,Z 1162.871,A -85,B 0,C 180,E1 19807.151,E2 19807.151} C_VEL
LIN {X 0,Y 409.308,Z 1168.429,A -85,B 0,C 180,E1 19804.678,E2 19804.678} C_VEL
LIN {X 0,Y 409.179,Z 1172.087,A -85,B 0,C 180,E1 19802.241,E2 19802.241} C_VEL
LIN {X 0,Y 409.151,Z 1173.945,A -85,B 0,C 180,E1 19799.86,E2 19799.86} C_VEL
LIN {X 0,Y 409.259,Z 1174.154,A -85,B 0,C 180,E1 19797.34,E2 19797.34} C_VEL
LIN {X 0,Y 409.485,Z 1172.624,A -85,B 0,C 180,E1 19794.817,E2 19794.817} C_VEL
LIN {X 0,Y 409.886,Z 1169.4,A -85,B 0,C 180,E1 19792.431,E2 19792.431} C_VEL
LIN {X 0,Y 410.463,Z 1164.435,A -85,B 0,C 180,E1 19790.041,E2 19790.041} C_VEL
LIN {X 0,Y 411.307,Z 1157.901,A -85,B 0,C 180,E1 19787.752,E2 19787.752} C_VEL
LIN {X 0,Y 412.414,Z 1149.524,A -85,B 0,C 180,E1 19785.54,E2 19785.54} C_VEL
LIN {X 0,Y 413.765,Z 1139.425,A -85,B 0,C 180,E1 19783.433,E2 19783.433} C_VEL
LIN {X 0,Y 415.155,Z 1128.506,A -85,B 0,C 180,E1 19781.607,E2 19781.607} C_VEL
LIN {X 0,Y 416.627,Z 1116.067,A -85,B 0,C 180,E1 19779.929,E2 19779.929} C_VEL
LIN {X 0,Y 418.051,Z 1102.653,A -85,B 0,C 180,E1 19778.462,E2 19778.462} C_VEL
LIN {X 0,Y 419.319,Z 1088.145,A -85,B 0,C 180,E1 19777.203,E2 19777.203} C_VEL
LIN {X 0,Y 420.351,Z 1072.623,A -85,B 0,C 180,E1 19776.149,E2 19776.149} C_VEL
LIN {X 0,Y 421.098,Z 1056.663,A -85,B 0,C 180,E1 19775.336,E2 19775.336} C_VEL
LIN {X 0,Y 421.676,Z 1034.565,A -85,B 0,C 180,E1 19774.575,E2 19774.575} C_VEL
LIN {X 0,Y 424.864,Z 988.651,A -85,B 0,C 180,E1 19773.157,E2 19773.157} C_VEL
LIN {X 0,Y 433.865,Z 901.639,A -85,B 0,C 180,E1 19770.375,E2 19770.375} C_VEL
LIN {X 0,Y 443.584,Z 882.198,A -85,B 0,C 180,E1 19768.962,E2 19768.962} C_VEL
LIN {X 0,Y 451.366,Z 863.032,A -85,B 0,C 180,E1 19766.373,E2 19766.373} C_VEL
LIN {X 0,Y 459.793,Z 848.178,A -85,B 0,C 180,E1 19764.2,E2 19764.2} C_VEL
LIN {X 0,Y 460.039,Z 847.816,A -85,B 0,C 180,E1 19764.11,E2 19764.11} C_VEL
LIN {X 0,Y 455.75,Z 855.874,A -85,B 0,C 180,E1 19762.577,E2 19762.577} C_VEL
LIN {X 0,Y 453.671,Z 864.062,A -85,B 0,C 180,E1 19761.016,E2 19761.016} C_VEL
LIN {X 0,Y 453.787,Z 872.492,A -85,B 0,C 180,E1 19759.459,E2 19759.459} C_VEL
LIN {X 0,Y 456.149,Z 881.424,A -85,B 0,C 180,E1 19757.876,E2 19757.876} C_VEL
LIN {X 0,Y 460.644,Z 890.455,A -85,B 0,C 180,E1 19756.351,E2 19756.351} C_VEL
LIN {X 0,Y 467.743,Z 900.124,A -85,B 0,C 180,E1 19754.791,E2 19754.791} C_VEL
LIN {X 0,Y 476.994,Z 909.519,A -85,B 0,C 180,E1 19753.334,E2 19753.334} C_VEL
LIN {X 0,Y 478.693,Z 911.157,A -85,B 0,C 180,E1 19753.1,E2 19753.1} C_VEL
LIN {X 0,Y 466.512,Z 932.239,A -85,B 0,C 180,E1 19752.548,E2 19752.548} C_VEL
LIN {X 0,Y 457.754,Z 950.191,A -85,B 0,C 180,E1 19751.943,E2 19751.943} C_VEL
LIN {X 0,Y 453.011,Z 960.874,A -85,B 0,C 180,E1 19751.54,E2 19751.54} C_VEL
LIN {X 0,Y 445.139,Z 978.008,A -85,B 0,C 180,E1 19750.902,E2 19750.902} C_VEL
LIN {X 0,Y 437.75,Z 998.336,A -85,B 0,C 180,E1 19750.025,E2 19750.025} C_VEL
LIN {X 0,Y 434.127,Z 1024.293,A -85,B 0,C 180,E1 19749.727,E2 19749.727} C_VEL
LIN {X 0,Y 432.695,Z 1050.697,A -85,B 0,C 180,E1 19749.107,E2 19749.107} C_VEL
LIN {X 0,Y 430.561,Z 1077.964,A -85,B 0,C 180,E1 19748.224,E2 19748.224} C_VEL
LIN {X 0,Y 428.407,Z 1101.972,A -85,B 0,C 180,E1 19747.192,E2 19747.192} C_VEL
LIN {X 0,Y 426.123,Z 1125.643,A -85,B 0,C 180,E1 19745.917,E2 19745.917} C_VEL
LIN {X 0,Y 423.77,Z 1148.653,A -85,B 0,C 180,E1 19744.409,E2 19744.409} C_VEL
LIN {X 0,Y 421.491,Z 1169.918,A -85,B 0,C 180,E1 19742.743,E2 19742.743} C_VEL
LIN {X 0,Y 419.19,Z 1190.445,A -85,B 0,C 180,E1 19740.832,E2 19740.832} C_VEL
LIN {X 0,Y 416.962,Z 1209.596,A -85,B 0,C 180,E1 19738.738,E2 19738.738} C_VEL
LIN {X 0,Y 414.936,Z 1227.169,A -85,B 0,C 180,E1 19736.474,E2 19736.474} C_VEL
LIN {X 0,Y 413.062,Z 1243.461,A -85,B 0,C 180,E1 19733.996,E2 19733.996} C_VEL
LIN {X 0,Y 411.485,Z 1257.919,A -85,B 0,C 180,E1 19731.376,E2 19731.376} C_VEL
LIN {X 0,Y 410.247,Z 1270.006,A -85,B 0,C 180,E1 19728.767,E2 19728.767} C_VEL
LIN {X 0,Y 409.382,Z 1279.995,A -85,B 0,C 180,E1 19726.167,E2 19726.167} C_VEL
LIN {X 0,Y 408.759,Z 1288.23,A -85,B 0,C 180,E1 19723.582,E2 19723.582} C_VEL
LIN {X 0,Y 408.377,Z 1295.144,A -85,B 0,C 180,E1 19720.867,E2 19720.867} C_VEL
LIN {X 0,Y 408.168,Z 1300.652,A -85,B 0,C 180,E1 19718.027,E2 19718.027} C_VEL
LIN {X 0,Y 408.089,Z 1304.266,A -85,B 0,C 180,E1 19715.343,E2 19715.343} C_VEL
LIN {X 0,Y 408.061,Z 1306.455,A -85,B 0,C 180,E1 19712.669,E2 19712.669} C_VEL
LIN {X 0,Y 408.057,Z 1307.208,A -85,B 0,C 180,E1 19709.72,E2 19709.72} C_VEL
LIN {X 0,Y 408.053,Z 1306.285,A -85,B 0,C 180,E1 19706.911,E2 19706.911} C_VEL
LIN {X 0,Y 408.067,Z 1304.17,A -85,B 0,C 180,E1 19704.376,E2 19704.376} C_VEL
LIN {X 0,Y 408.135,Z 1300.548,A -85,B 0,C 180,E1 19701.69,E2 19701.69} C_VEL
LIN {X 0,Y 408.364,Z 1294.822,A -85,B 0,C 180,E1 19698.705,E2 19698.705} C_VEL
LIN {X 0,Y 408.775,Z 1287.987,A -85,B 0,C 180,E1 19695.987,E2 19695.987} C_VEL
LIN {X 0,Y 409.473,Z 1279.519,A -85,B 0,C 180,E1 19693.254,E2 19693.254} C_VEL
LIN {X 0,Y 410.637,Z 1267.986,A -85,B 0,C 180,E1 19690.218,E2 19690.218} C_VEL
LIN {X 0,Y 412.043,Z 1256.052,A -85,B 0,C 180,E1 19687.597,E2 19687.597} C_VEL
LIN {X 0,Y 414.011,Z 1241.292,A -85,B 0,C 180,E1 19684.847,E2 19684.847} C_VEL
LIN {X 0,Y 416.376,Z 1224.634,A -85,B 0,C 180,E1 19682.235,E2 19682.235} C_VEL
LIN {X 0,Y 419.057,Z 1206.497,A -85,B 0,C 180,E1 19679.827,E2 19679.827} C_VEL
LIN {X 0,Y 421.663,Z 1188.781,A -85,B 0,C 180,E1 19677.835,E2 19677.835} C_VEL
LIN {X 0,Y 424.474,Z 1169.67,A -85,B 0,C 180,E1 19675.992,E2 19675.992} C_VEL
LIN {X 0,Y 427.126,Z 1150.74,A -85,B 0,C 180,E1 19674.454,E2 19674.454} C_VEL
LIN {X 0,Y 429.916,Z 1129.707,A -85,B 0,C 180,E1 19673.015,E2 19673.015} C_VEL
LIN {X 0,Y 432.596,Z 1107.647,A -85,B 0,C 180,E1 19671.798,E2 19671.798} C_VEL
LIN {X 0,Y 434.939,Z 1085.059,A -85,B 0,C 180,E1 19670.827,E2 19670.827} C_VEL
LIN {X 0,Y 436.927,Z 1062.119,A -85,B 0,C 180,E1 19670.1,E2 19670.1} C_VEL
LIN {X 0,Y 438.337,Z 1035.253,A -85,B 0,C 180,E1 19669.495,E2 19669.495} C_VEL
LIN {X 0,Y 439.508,Z 1017.92,A -85,B 0,C 180,E1 19669.205,E2 19669.205} C_VEL
LIN {X 0,Y 440.061,Z 1013.466,A -85,B 0,C 180,E1 19669.13,E2 19669.13} C_VEL
LIN {X 0,Y 450.106,Z 986.441,A -85,B 0,C 180,E1 19667.868,E2 19667.868} C_VEL
LIN {X 0,Y 457.897,Z 969.395,A -85,B 0,C 180,E1 19667.228,E2 19667.228} C_VEL
LIN {X 0,Y 461.985,Z 960.951,A -85,B 0,C 180,E1 19666.936,E2 19666.936} C_VEL
LIN {X 0,Y 470.443,Z 942.993,A -85,B 0,C 180,E1 19666.312,E2 19666.312} C_VEL
LIN {X 0,Y 481.803,Z 922.562,A -85,B 0,C 180,E1 19665.792,E2 19665.792} C_VEL
LIN {X 0,Y 485.053,Z 916.916,A -85,B 0,C 180,E1 19665.666,E2 19665.666} C_VEL
LIN {X 0,Y 475.389,Z 906.984,A -85,B 0,C 180,E1 19663.953,E2 19663.953} C_VEL
LIN {X 0,Y 467.31,Z 895.662,A -85,B 0,C 180,E1 19662.208,E2 19662.208} C_VEL
LIN {X 0,Y 460.735,Z 882.475,A -85,B 0,C 180,E1 19660.385,E2 19660.385} C_VEL
LIN {X 0,Y 456.01,Z 868.131,A -85,B 0,C 180,E1 19658.594,E2 19658.594} C_VEL
LIN {X 0,Y 453.042,Z 852.365,A -85,B 0,C 180,E1 19656.812,E2 19656.812} C_VEL
LIN {X 0,Y 451.862,Z 834.265,A -85,B 0,C 180,E1 19654.966,E2 19654.966} C_VEL
LIN {X 0,Y 452.641,Z 814.378,A -85,B 0,C 180,E1 19653.157,E2 19653.157} C_VEL
LIN {X 0,Y 458.032,Z 771.567,A -85,B 0,C 180,E1 19649.64,E2 19649.64} C_VEL
LIN {X 0,Y 448.816,Z 753.994,A -85,B 0,C 180,E1 19646.316,E2 19646.316} C_VEL
LIN {X 0,Y 440.221,Z 737.964,A -85,B 0,C 180,E1 19642.995,E2 19642.995} C_VEL
LIN {X 0,Y 432.223,Z 723.71,A -85,B 0,C 180,E1 19639.739,E2 19639.739} C_VEL
LIN {X 0,Y 425.992,Z 712.953,A -85,B 0,C 180,E1 19637.061,E2 19637.061} C_VEL
LIN {X 0,Y 423.419,Z 708.443,A -85,B 0,C 180,E1 19635.897,E2 19635.897} C_VEL
LIN {X 0,Y 420.592,Z 703.572,A -85,B 0,C 180,E1 19634.595,E2 19634.595} C_VEL
LIN {X 0,Y 417.862,Z 698.809,A -85,B 0,C 180,E1 19633.28,E2 19633.28} C_VEL
LIN {X 0,Y 415.694,Z 695.015,A -85,B 0,C 180,E1 19632.22,E2 19632.22} C_VEL
LIN {X 0,Y 412.733,Z 690.066,A -85,B 0,C 180,E1 19630.75,E2 19630.75} C_VEL
LIN {X 0,Y 411.985,Z 688.648,A -85,B 0,C 180,E1 19630.346,E2 19630.346} C_VEL
LIN {X 0,Y 410.008,Z 685.867,A -85,B 0,C 180,E1 19629.403,E2 19629.403} C_VEL
LIN {X 0,Y 409.439,Z 683.731,A -85,B 0,C 180,E1 19628.85,E2 19628.85} C_VEL
LIN {X 0,Y 409.44,Z 683.731,A -85,B 0,C 180,E1 19624.913,E2 19624.913} C_VEL
LIN {X 0,Y 409.445,Z 683.73,A -85,B 0,C 180,E1 19620.839,E2 19620.839} C_VEL
LIN {X 0,Y 409.434,Z 683.736,A -85,B 0,C 180,E1 19616.92,E2 19616.92} C_VEL
LIN {X 0,Y 409.447,Z 683.734,A -85,B 0,C 180,E1 19612.986,E2 19612.986} C_VEL
LIN {X 0,Y 409.437,Z 683.731,A -85,B 0,C 180,E1 19609.016,E2 19609.016} C_VEL
LIN {X 0,Y 409.433,Z 683.735,A -85,B 0,C 180,E1 19605.142,E2 19605.142} C_VEL
LIN {X 0,Y 409.434,Z 683.721,A -85,B 0,C 180,E1 19601.342,E2 19601.342} C_VEL
LIN {X 0,Y 409.433,Z 683.727,A -85,B 0,C 180,E1 19597.606,E2 19597.606} C_VEL
LIN {X 0,Y 409.438,Z 683.722,A -85,B 0,C 180,E1 19593.664,E2 19593.664} C_VEL
LIN {X 0,Y 409.426,Z 683.689,A -85,B 0,C 180,E1 19589.796,E2 19589.796} C_VEL
LIN {X 0,Y 409.438,Z 683.696,A -85,B 0,C 180,E1 19585.877,E2 19585.877} C_VEL
LIN {X 0,Y 409.448,Z 683.795,A -85,B 0,C 180,E1 19582.122,E2 19582.122} C_VEL
LIN {X 0,Y 410.612,Z 687.003,A -85,B 0,C 180,E1 19581.615,E2 19581.615} C_VEL
LIN {X 0,Y 412.219,Z 689.276,A -85,B 0,C 180,E1 19581.131,E2 19581.131} C_VEL
LIN {X 0,Y 414.342,Z 693.115,A -85,B 0,C 180,E1 19580.426,E2 19580.426} C_VEL
LIN {X 0,Y 421.961,Z 707.785,A -85,B 0,C 180,E1 19577.888,E2 19577.888} C_VEL
LIN {X 0,Y 429.611,Z 723.93,A -85,B 0,C 180,E1 19575.343,E2 19575.343} C_VEL
LIN {X 0,Y 437.41,Z 742.643,A -85,B 0,C 180,E1 19572.7,E2 19572.7} C_VEL
LIN {X 0,Y 438.292,Z 745.567,A -85,B 0,C 180,E1 19572.342,E2 19572.342} C_VEL
LIN {X 0,Y 436.769,Z 774.751,A -85,B 0,C 180,E1 19570.209,E2 19570.209} C_VEL
LIN {X 0,Y 439.97,Z 798.727,A -85,B 0,C 180,E1 19569.351,E2 19569.351} C_VEL
LIN {X 0,Y 433.431,Z 1034.384,A -85,B 0,C 180,E1 19565.168,E2 19565.168} C_VEL
LIN {X 0,Y 432.59,Z 1051.974,A -85,B 0,C 180,E1 19564.697,E2 19564.697} C_VEL
LIN {X 0,Y 431.2,Z 1059.5,A -85,B 0,C 180,E1 19564.524,E2 19564.524} C_VEL
LIN {X 0,Y 424.859,Z 1078.405,A -85,B 0,C 180,E1 19564.188,E2 19564.188} C_VEL
LIN {X 0,Y 423.284,Z 1085.653,A -85,B 0,C 180,E1 19563.891,E2 19563.891} C_VEL
LIN {X 0,Y 421.164,Z 1104.289,A -85,B 0,C 180,E1 19562.77,E2 19562.77} C_VEL
LIN {X 0,Y 418.667,Z 1122.803,A -85,B 0,C 180,E1 19561.373,E2 19561.373} C_VEL
LIN {X 0,Y 416.107,Z 1139.627,A -85,B 0,C 180,E1 19559.827,E2 19559.827} C_VEL
LIN {X 0,Y 413.359,Z 1156.3,A -85,B 0,C 180,E1 19557.985,E2 19557.985} C_VEL
LIN {X 0,Y 410.539,Z 1172.407,A -85,B 0,C 180,E1 19555.845,E2 19555.845} C_VEL
LIN {X 0,Y 407.973,Z 1186.806,A -85,B 0,C 180,E1 19553.545,E2 19553.545} C_VEL
LIN {X 0,Y 405.849,Z 1198.958,A -85,B 0,C 180,E1 19551.232,E2 19551.232} C_VEL
LIN {X 0,Y 403.945,Z 1210.398,A -85,B 0,C 180,E1 19548.62,E2 19548.62} C_VEL
LIN {X 0,Y 402.447,Z 1220.294,A -85,B 0,C 180,E1 19545.859,E2 19545.859} C_VEL
LIN {X 0,Y 401.354,Z 1228.609,A -85,B 0,C 180,E1 19542.956,E2 19542.956} C_VEL
LIN {X 0,Y 400.685,Z 1235.025,A -85,B 0,C 180,E1 19540.059,E2 19540.059} C_VEL
LIN {X 0,Y 400.322,Z 1239.717,A -85,B 0,C 180,E1 19537.173,E2 19537.173} C_VEL
LIN {X 0,Y 400.154,Z 1242.918,A -85,B 0,C 180,E1 19534.155,E2 19534.155} C_VEL
LIN {X 0,Y 400.099,Z 1244.407,A -85,B 0,C 180,E1 19531.288,E2 19531.288} C_VEL
LIN {X 0,Y 400.1,Z 1244.377,A -85,B 0,C 180,E1 19528.408,E2 19528.408} C_VEL
LIN {X 0,Y 400.164,Z 1242.751,A -85,B 0,C 180,E1 19525.528,E2 19525.528} C_VEL
LIN {X 0,Y 400.326,Z 1239.645,A -85,B 0,C 180,E1 19522.681,E2 19522.681} C_VEL
LIN {X 0,Y 400.693,Z 1234.913,A -85,B 0,C 180,E1 19519.795,E2 19519.795} C_VEL
LIN {X 0,Y 401.368,Z 1228.505,A -85,B 0,C 180,E1 19516.915,E2 19516.915} C_VEL
LIN {X 0,Y 402.449,Z 1220.286,A -85,B 0,C 180,E1 19514.046,E2 19514.046} C_VEL
LIN {X 0,Y 403.986,Z 1210.183,A -85,B 0,C 180,E1 19511.231,E2 19511.231} C_VEL
LIN {X 0,Y 405.909,Z 1198.651,A -85,B 0,C 180,E1 19508.61,E2 19508.61} C_VEL
LIN {X 0,Y 408.041,Z 1186.481,A -85,B 0,C 180,E1 19506.305,E2 19506.305} C_VEL
LIN {X 0,Y 410.533,Z 1172.505,A -85,B 0,C 180,E1 19504.076,E2 19504.076} C_VEL
LIN {X 0,Y 413.352,Z 1156.411,A -85,B 0,C 180,E1 19501.934,E2 19501.934} C_VEL
LIN {X 0,Y 416.099,Z 1139.754,A -85,B 0,C 180,E1 19500.092,E2 19500.092} C_VEL
LIN {X 0,Y 418.664,Z 1122.955,A -85,B 0,C 180,E1 19498.545,E2 19498.545} C_VEL
LIN {X 0,Y 421.162,Z 1104.468,A -85,B 0,C 180,E1 19497.148,E2 19497.148} C_VEL
LIN {X 0,Y 423.405,Z 1084.783,A -85,B 0,C 180,E1 19495.967,E2 19495.967} C_VEL
LIN {X 0,Y 425.151,Z 1065.292,A -85,B 0,C 180,E1 19495.064,E2 19495.064} C_VEL
LIN {X 0,Y 426.471,Z 1044.91,A -85,B 0,C 180,E1 19494.371,E2 19494.371} C_VEL
LIN {X 0,Y 427.405,Z 1021.03,A -85,B 0,C 180,E1 19493.847,E2 19493.847} C_VEL
LIN {X 0,Y 433.521,Z 808.564,A -85,B 0,C 180,E1 19490.048,E2 19490.048} C_VEL
LIN {X 0,Y 426.676,Z 776.622,A -85,B 0,C 180,E1 19488.538,E2 19488.538} C_VEL
LIN {X 0,Y 428.411,Z 749.341,A -85,B 0,C 180,E1 19485.606,E2 19485.606} C_VEL
LIN {X 0,Y 422.51,Z 731.933,A -85,B 0,C 180,E1 19482.595,E2 19482.595} C_VEL
LIN {X 0,Y 420.998,Z 728.288,A -85,B 0,C 180,E1 19481.879,E2 19481.879} C_VEL
LIN {X 0,Y 427.657,Z 745.628,A -85,B 0,C 180,E1 19478.971,E2 19478.971} C_VEL
LIN {X 0,Y 428.126,Z 747.725,A -85,B 0,C 180,E1 19478.671,E2 19478.671} C_VEL
LIN {X 0,Y 424.052,Z 785.833,A -85,B 0,C 180,E1 19474.793,E2 19474.793} C_VEL
LIN {X 0,Y 419.976,Z 827.423,A -85,B 0,C 180,E1 19470.63,E2 19470.63} C_VEL
LIN {X 0,Y 417.002,Z 862.197,A -85,B 0,C 180,E1 19467.228,E2 19467.228} C_VEL
LIN {X 0,Y 418.21,Z 871.996,A -85,B 0,C 180,E1 19466.883,E2 19466.883} C_VEL
LIN {X 0,Y 412.36,Z 1033.085,A -85,B 0,C 180,E1 19463.265,E2 19463.265} C_VEL
LIN {X 0,Y 411.687,Z 1050.738,A -85,B 0,C 180,E1 19462.603,E2 19462.603} C_VEL
LIN {X 0,Y 410.727,Z 1067.574,A -85,B 0,C 180,E1 19461.717,E2 19461.717} C_VEL
LIN {X 0,Y 409.529,Z 1083.898,A -85,B 0,C 180,E1 19460.584,E2 19460.584} C_VEL
LIN {X 0,Y 408.187,Z 1099.105,A -85,B 0,C 180,E1 19459.234,E2 19459.234} C_VEL
LIN {X 0,Y 406.755,Z 1113.921,A -85,B 0,C 180,E1 19457.599,E2 19457.599} C_VEL
LIN {X 0,Y 405.456,Z 1126.541,A -85,B 0,C 180,E1 19455.886,E2 19455.886} C_VEL
LIN {X 0,Y 404.195,Z 1138.483,A -85,B 0,C 180,E1 19453.884,E2 19453.884} C_VEL
LIN {X 0,Y 403.127,Z 1148.867,A -85,B 0,C 180,E1 19451.735,E2 19451.735} C_VEL
LIN {X 0,Y 402.352,Z 1157.198,A -85,B 0,C 180,E1 19449.585,E2 19449.585} C_VEL
LIN {X 0,Y 401.779,Z 1164.457,A -85,B 0,C 180,E1 19447.148,E2 19447.148} C_VEL
LIN {X 0,Y 401.43,Z 1169.809,A -85,B 0,C 180,E1 19444.715,E2 19444.715} C_VEL
LIN {X 0,Y 401.298,Z 1173.425,A -85,B 0,C 180,E1 19442.285,E2 19442.285} C_VEL
LIN {X 0,Y 401.273,Z 1175.339,A -85,B 0,C 180,E1 19439.858,E2 19439.858} C_VEL
LIN {X 0,Y 401.396,Z 1175.602,A -85,B 0,C 180,E1 19437.288,E2 19437.288} C_VEL
LIN {X 0,Y 401.65,Z 1174.118,A -85,B 0,C 180,E1 19434.715,E2 19434.715} C_VEL
LIN {X 0,Y 402.096,Z 1170.95,A -85,B 0,C 180,E1 19432.283,E2 19432.283} C_VEL
LIN {X 0,Y 402.734,Z 1166.05,A -85,B 0,C 180,E1 19429.848,E2 19429.848} C_VEL
LIN {X 0,Y 403.637,Z 1159.693,A -85,B 0,C 180,E1 19427.555,E2 19427.555} C_VEL
LIN {X 0,Y 404.853,Z 1151.263,A -85,B 0,C 180,E1 19425.264,E2 19425.264} C_VEL
LIN {X 0,Y 406.311,Z 1141.278,A -85,B 0,C 180,E1 19423.12,E2 19423.12} C_VEL
LIN {X 0,Y 407.787,Z 1130.426,A -85,B 0,C 180,E1 19421.265,E2 19421.265} C_VEL
LIN {X 0,Y 409.439,Z 1117.569,A -85,B 0,C 180,E1 19419.487,E2 19419.487} C_VEL
LIN {X 0,Y 410.954,Z 1104.16,A -85,B 0,C 180,E1 19417.996,E2 19417.996} C_VEL
LIN {X 0,Y 412.381,Z 1088.795,A -85,B 0,C 180,E1 19416.646,E2 19416.646} C_VEL
LIN {X 0,Y 413.425,Z 1074.354,A -85,B 0,C 180,E1 19415.648,E2 19415.648} C_VEL
LIN {X 0,Y 414.237,Z 1057.561,A -85,B 0,C 180,E1 19414.785,E2 19414.785} C_VEL
LIN {X 0,Y 415.243,Z 1030.376,A -85,B 0,C 180,E1 19413.822,E2 19413.822} C_VEL
LIN {X 0,Y 419.797,Z 979.244,A -85,B 0,C 180,E1 19412.119,E2 19412.119} C_VEL
LIN {X 0,Y 428.505,Z 905.941,A -85,B 0,C 180,E1 19409.657,E2 19409.657} C_VEL
LIN {X 0,Y 439.169,Z 885.554,A -85,B 0,C 180,E1 19408.193,E2 19408.193} C_VEL
LIN {X 0,Y 446.912,Z 868.51,A -85,B 0,C 180,E1 19405.837,E2 19405.837} C_VEL
LIN {X 0,Y 454.114,Z 856.601,A -85,B 0,C 180,E1 19404.033,E2 19404.033} C_VEL
LIN {X 0,Y 450.209,Z 864.492,A -85,B 0,C 180,E1 19402.453,E2 19402.453} C_VEL
LIN {X 0,Y 448.529,Z 872.442,A -85,B 0,C 180,E1 19400.875,E2 19400.875} C_VEL
LIN {X 0,Y 449.005,Z 880.776,A -85,B 0,C 180,E1 19399.273,E2 19399.273} C_VEL
LIN {X 0,Y 451.7,Z 889.478,A -85,B 0,C 180,E1 19397.674,E2 19397.674} C_VEL
LIN {X 0,Y 456.325,Z 898.023,A -85,B 0,C 180,E1 19396.181,E2 19396.181} C_VEL
LIN {X 0,Y 463.546,Z 907.405,A -85,B 0,C 180,E1 19394.619,E2 19394.619} C_VEL
LIN {X 0,Y 469.727,Z 914.037,A -85,B 0,C 180,E1 19393.583,E2 19393.583} C_VEL
LIN {X 0,Y 458.128,Z 934.846,A -85,B 0,C 180,E1 19393.019,E2 19393.019} C_VEL
LIN {X 0,Y 449.568,Z 953.195,A -85,B 0,C 180,E1 19392.368,E2 19392.368} C_VEL
LIN {X 0,Y 438.414,Z 977.478,A -85,B 0,C 180,E1 19391.468,E2 19391.468} C_VEL
LIN {X 0,Y 431.907,Z 995.194,A -85,B 0,C 180,E1 19390.695,E2 19390.695} C_VEL
LIN {X 0,Y 427.786,Z 1023.374,A -85,B 0,C 180,E1 19390.376,E2 19390.376} C_VEL
LIN {X 0,Y 426.155,Z 1048.412,A -85,B 0,C 180,E1 19389.76,E2 19389.76} C_VEL
LIN {X 0,Y 423.846,Z 1075.619,A -85,B 0,C 180,E1 19388.85,E2 19388.85} C_VEL
LIN {X 0,Y 421.379,Z 1100.576,A -85,B 0,C 180,E1 19387.748,E2 19387.748} C_VEL
LIN {X 0,Y 418.836,Z 1125.12,A -85,B 0,C 180,E1 19386.387,E2 19386.387} C_VEL
LIN {X 0,Y 416.363,Z 1147.817,A -85,B 0,C 180,E1 19384.858,E2 19384.858} C_VEL
LIN {X 0,Y 413.865,Z 1169.638,A -85,B 0,C 180,E1 19383.093,E2 19383.093} C_VEL
LIN {X 0,Y 411.326,Z 1191.262,A -85,B 0,C 180,E1 19381.02,E2 19381.02} C_VEL
LIN {X 0,Y 409.096,Z 1209.621,A -85,B 0,C 180,E1 19378.943,E2 19378.943} C_VEL
LIN {X 0,Y 407.077,Z 1226.509,A -85,B 0,C 180,E1 19376.711,E2 19376.711} C_VEL
LIN {X 0,Y 405.26,Z 1241.897,A -85,B 0,C 180,E1 19374.333,E2 19374.333} C_VEL
LIN {X 0,Y 403.623,Z 1256.487,A -85,B 0,C 180,E1 19371.661,E2 19371.661} C_VEL
LIN {X 0,Y 402.347,Z 1268.653,A -85,B 0,C 180,E1 19368.999,E2 19368.999} C_VEL
LIN {X 0,Y 401.462,Z 1278.754,A -85,B 0,C 180,E1 19366.346,E2 19366.346} C_VEL
LIN {X 0,Y 400.797,Z 1287.465,A -85,B 0,C 180,E1 19363.563,E2 19363.563} C_VEL
LIN {X 0,Y 400.433,Z 1294.289,A -85,B 0,C 180,E1 19360.794,E2 19360.794} C_VEL
LIN {X 0,Y 400.237,Z 1299.752,A -85,B 0,C 180,E1 19357.898,E2 19357.898} C_VEL
LIN {X 0,Y 400.163,Z 1303.458,A -85,B 0,C 180,E1 19355.018,E2 19355.018} C_VEL
LIN {X 0,Y 400.156,Z 1305.592,A -85,B 0,C 180,E1 19352.005,E2 19352.005} C_VEL
LIN {X 0,Y 400.137,Z 1305.961,A -85,B 0,C 180,E1 19349.142,E2 19349.142} C_VEL
LIN {X 0,Y 400.128,Z 1304.854,A -85,B 0,C 180,E1 19346.419,E2 19346.419} C_VEL
LIN {X 0,Y 400.147,Z 1302.204,A -85,B 0,C 180,E1 19343.545,E2 19343.545} C_VEL
LIN {X 0,Y 400.24,Z 1297.677,A -85,B 0,C 180,E1 19340.511,E2 19340.511} C_VEL
LIN {X 0,Y 400.522,Z 1291.892,A -85,B 0,C 180,E1 19337.75,E2 19337.75} C_VEL
LIN {X 0,Y 401.002,Z 1284.667,A -85,B 0,C 180,E1 19334.971,E2 19334.971} C_VEL
LIN {X 0,Y 401.874,Z 1275.113,A -85,B 0,C 180,E1 19332.031,E2 19332.031} C_VEL
LIN {X 0,Y 403.109,Z 1264.089,A -85,B 0,C 180,E1 19329.226,E2 19329.226} C_VEL
LIN {X 0,Y 404.912,Z 1250.195,A -85,B 0,C 180,E1 19326.266,E2 19326.266} C_VEL
LIN {X 0,Y 407.161,Z 1234.408,A -85,B 0,C 180,E1 19323.454,E2 19323.454} C_VEL
LIN {X 0,Y 409.767,Z 1217.221,A -85,B 0,C 180,E1 19320.872,E2 19320.872} C_VEL
LIN {X 0,Y 412.644,Z 1198.754,A -85,B 0,C 180,E1 19318.53,E2 19318.53} C_VEL
LIN {X 0,Y 415.854,Z 1178.112,A -85,B 0,C 180,E1 19316.337,E2 19316.337} C_VEL
LIN {X 0,Y 418.728,Z 1158.995,A -85,B 0,C 180,E1 19314.612,E2 19314.612} C_VEL
LIN {X 0,Y 421.867,Z 1137.226,A -85,B 0,C 180,E1 19312.988,E2 19312.988} C_VEL
LIN {X 0,Y 424.705,Z 1115.406,A -85,B 0,C 180,E1 19311.66,E2 19311.66} C_VEL
LIN {X 0,Y 427.375,Z 1092.698,A -85,B 0,C 180,E1 19310.567,E2 19310.567} C_VEL
LIN {X 0,Y 429.688,Z 1069.471,A -85,B 0,C 180,E1 19309.719,E2 19309.719} C_VEL
LIN {X 0,Y 431.29,Z 1046.46,A -85,B 0,C 180,E1 19309.123,E2 19309.123} C_VEL
LIN {X 0,Y 432.671,Z 1021.272,A -85,B 0,C 180,E1 19308.634,E2 19308.634} C_VEL
LIN {X 0,Y 433.747,Z 1012.303,A -85,B 0,C 180,E1 19308.492,E2 19308.492} C_VEL
LIN {X 0,Y 444.331,Z 984.392,A -85,B 0,C 180,E1 19307.19,E2 19307.19} C_VEL
LIN {X 0,Y 452.689,Z 966.579,A -85,B 0,C 180,E1 19306.528,E2 19306.528} C_VEL
LIN {X 0,Y 456.701,Z 958.146,A -85,B 0,C 180,E1 19306.227,E2 19306.227} C_VEL
LIN {X 0,Y 465.315,Z 940.314,A -85,B 0,C 180,E1 19305.62,E2 19305.62} C_VEL
LIN {X 0,Y 476.581,Z 919.997,A -85,B 0,C 180,E1 19305.099,E2 19305.099} C_VEL
LIN {X 0,Y 466.874,Z 908.943,A -85,B 0,C 180,E1 19303.26,E2 19303.26} C_VEL
LIN {X 0,Y 459.521,Z 897.515,A -85,B 0,C 180,E1 19301.541,E2 19301.541} C_VEL
LIN {X 0,Y 453.33,Z 883.804,A -85,B 0,C 180,E1 19299.67,E2 19299.67} C_VEL
LIN {X 0,Y 449.033,Z 868.99,A -85,B 0,C 180,E1 19297.839,E2 19297.839} C_VEL
LIN {X 0,Y 446.481,Z 852.701,A -85,B 0,C 180,E1 19296.012,E2 19296.012} C_VEL
LIN {X 0,Y 445.693,Z 833.865,A -85,B 0,C 180,E1 19294.114,E2 19294.114} C_VEL
LIN {X 0,Y 447.061,Z 812.123,A -85,B 0,C 180,E1 19292.16,E2 19292.16} C_VEL
LIN {X 0,Y 451.954,Z 775.82,A -85,B 0,C 180,E1 19289.16,E2 19289.16} C_VEL
LIN {X 0,Y 442.257,Z 757.169,A -85,B 0,C 180,E1 19285.572,E2 19285.572} C_VEL
LIN {X 0,Y 433.668,Z 741.41,A -85,B 0,C 180,E1 19282.217,E2 19282.217} C_VEL
LIN {X 0,Y 426.645,Z 728.84,A -85,B 0,C 180,E1 19279.295,E2 19279.295} C_VEL
LIN {X 0,Y 421.021,Z 719.009,A -85,B 0,C 180,E1 19276.841,E2 19276.841} C_VEL
LIN {X 0,Y 418.168,Z 714.045,A -85,B 0,C 180,E1 19275.533,E2 19275.533} C_VEL
LIN {X 0,Y 415.637,Z 709.616,A -85,B 0,C 180,E1 19274.346,E2 19274.346} C_VEL
LIN {X 0,Y 412.866,Z 704.831,A -85,B 0,C 180,E1 19273.016,E2 19273.016} C_VEL
LIN {X 0,Y 409.885,Z 699.736,A -85,B 0,C 180,E1 19271.538,E2 19271.538} C_VEL
LIN {X 0,Y 407.785,Z 695.986,A -85,B 0,C 180,E1 19270.453,E2 19270.453} C_VEL
LIN {X 0,Y 404.847,Z 691.189,A -85,B 0,C 180,E1 19268.951,E2 19268.951} C_VEL
LIN {X 0,Y 404.153,Z 689.74,A -85,B 0,C 180,E1 19268.536,E2 19268.536} C_VEL
LIN {X 0,Y 401.957,Z 686.57,A -85,B 0,C 180,E1 19267.432,E2 19267.432} C_VEL
LIN {X 0,Y 401.504,Z 684.719,A -85,B 0,C 180,E1 19266.937,E2 19266.937} C_VEL
LIN {X 0,Y 401.493,Z 684.721,A -85,B 0,C 180,E1 19262.997,E2 19262.997} C_VEL
LIN {X 0,Y 401.495,Z 684.724,A -85,B 0,C 180,E1 19259.144,E2 19259.144} C_VEL
LIN {X 0,Y 401.501,Z 684.723,A -85,B 0,C 180,E1 19255.143,E2 19255.143} C_VEL
LIN {X 0,Y 401.492,Z 684.72,A -85,B 0,C 180,E1 19251.262,E2 19251.262} C_VEL
LIN {X 0,Y 401.503,Z 684.721,A -85,B 0,C 180,E1 19247.341,E2 19247.341} C_VEL
LIN {X 0,Y 401.503,Z 684.722,A -85,B 0,C 180,E1 19243.358,E2 19243.358} C_VEL
LIN {X 0,Y 401.509,Z 684.72,A -85,B 0,C 180,E1 19239.291,E2 19239.291} C_VEL
LIN {X 0,Y 401.496,Z 684.722,A -85,B 0,C 180,E1 19235.268,E2 19235.268} C_VEL
LIN {X 0,Y 401.493,Z 684.662,A -85,B 0,C 180,E1 19231.273,E2 19231.273} C_VEL
LIN {X 0,Y 401.502,Z 684.721,A -85,B 0,C 180,E1 19227.289,E2 19227.289} C_VEL
LIN {X 0,Y 401.507,Z 684.829,A -85,B 0,C 180,E1 19223.406,E2 19223.406} C_VEL
LIN {X 0,Y 402.658,Z 687.954,A -85,B 0,C 180,E1 19222.886,E2 19222.886} C_VEL
LIN {X 0,Y 404.37,Z 690.273,A -85,B 0,C 180,E1 19222.357,E2 19222.357} C_VEL
LIN {X 0,Y 406.293,Z 693.914,A -85,B 0,C 180,E1 19221.672,E2 19221.672} C_VEL
LIN {X 0,Y 412.256,Z 704.843,A -85,B 0,C 180,E1 19219.641,E2 19219.641} C_VEL
LIN {X 0,Y 419.834,Z 720.012,A -85,B 0,C 180,E1 19217.068,E2 19217.068} C_VEL
LIN {X 0,Y 427.949,Z 738.461,A -85,B 0,C 180,E1 19214.275,E2 19214.275} C_VEL
LIN {X 0,Y 431.972,Z 749.091,A -85,B 0,C 180,E1 19212.835,E2 19212.835} C_VEL
LIN {X 0,Y 430.562,Z 775.376,A -85,B 0,C 180,E1 19210.908,E2 19210.908} C_VEL
LIN {X 0,Y 433.797,Z 800.091,A -85,B 0,C 180,E1 19210.004,E2 19210.004} C_VEL
LIN {X 0,Y 426.908,Z 1035.494,A -85,B 0,C 180,E1 19205.772,E2 19205.772} C_VEL
LIN {X 0,Y 425.74,Z 1056.767,A -85,B 0,C 180,E1 19205.162,E2 19205.162} C_VEL
LIN {X 0,Y 424.131,Z 1076.887,A -85,B 0,C 180,E1 19204.333,E2 19204.333} C_VEL
LIN {X 0,Y 423.284,Z 1085.653,A -85,B 0,C 180,E1 19203.891,E2 19203.891} C_VEL
LIN {X 0,Y 421.651,Z 1093.045,A -85,B 0,C 180,E1 19203.56,E2 19203.56} C_VEL
LIN {X 0,Y 414.466,Z 1110.932,A -85,B 0,C 180,E1 19202.859,E2 19202.859} C_VEL
LIN {X 0,Y 412.668,Z 1117.732,A -85,B 0,C 180,E1 19202.415,E2 19202.415} C_VEL
LIN {X 0,Y 410.125,Z 1134.525,A -85,B 0,C 180,E1 19200.957,E2 19200.957} C_VEL
LIN {X 0,Y 407.131,Z 1152.171,A -85,B 0,C 180,E1 19199.094,E2 19199.094} C_VEL
LIN {X 0,Y 404.247,Z 1168.008,A -85,B 0,C 180,E1 19197.071,E2 19197.071} C_VEL
LIN {X 0,Y 401.546,Z 1182.322,A -85,B 0,C 180,E1 19194.885,E2 19194.885} C_VEL
LIN {X 0,Y 399.111,Z 1195.231,A -85,B 0,C 180,E1 19192.537,E2 19192.537} C_VEL
LIN {X 0,Y 396.903,Z 1207.391,A -85,B 0,C 180,E1 19189.881,E2 19189.881} C_VEL
LIN {X 0,Y 395.203,Z 1217.458,A -85,B 0,C 180,E1 19187.217,E2 19187.217} C_VEL
LIN {X 0,Y 393.913,Z 1226.128,A -85,B 0,C 180,E1 19184.403,E2 19184.403} C_VEL
LIN {X 0,Y 393.022,Z 1233.323,A -85,B 0,C 180,E1 19181.445,E2 19181.445} C_VEL
LIN {X 0,Y 392.499,Z 1238.675,A -85,B 0,C 180,E1 19178.496,E2 19178.496} C_VEL
LIN {X 0,Y 392.239,Z 1242.372,A -85,B 0,C 180,E1 19175.558,E2 19175.558} C_VEL
LIN {X 0,Y 392.14,Z 1244.587,A -85,B 0,C 180,E1 19172.484,E2 19172.484} C_VEL
LIN {X 0,Y 392.118,Z 1245.158,A -85,B 0,C 180,E1 19169.561,E2 19169.561} C_VEL
LIN {X 0,Y 392.16,Z 1244.239,A -85,B 0,C 180,E1 19166.638,E2 19166.638} C_VEL
LIN {X 0,Y 392.287,Z 1241.711,A -85,B 0,C 180,E1 19163.707,E2 19163.707} C_VEL
LIN {X 0,Y 392.591,Z 1237.612,A -85,B 0,C 180,E1 19160.766,E2 19160.766} C_VEL
LIN {X 0,Y 393.223,Z 1231.51,A -85,B 0,C 180,E1 19157.667,E2 19157.667} C_VEL
LIN {X 0,Y 394.236,Z 1223.828,A -85,B 0,C 180,E1 19154.706,E2 19154.706} C_VEL
LIN {X 0,Y 395.67,Z 1214.649,A -85,B 0,C 180,E1 19151.891,E2 19151.891} C_VEL
LIN {X 0,Y 397.524,Z 1204.023,A -85,B 0,C 180,E1 19149.228,E2 19149.228} C_VEL
LIN {X 0,Y 399.761,Z 1191.958,A -85,B 0,C 180,E1 19146.722,E2 19146.722} C_VEL
LIN {X 0,Y 402.31,Z 1178.379,A -85,B 0,C 180,E1 19144.377,E2 19144.377} C_VEL
LIN {X 0,Y 405.015,Z 1163.825,A -85,B 0,C 180,E1 19142.269,E2 19142.269} C_VEL
LIN {X 0,Y 407.893,Z 1147.754,A -85,B 0,C 180,E1 19140.319,E2 19140.319} C_VEL
LIN {X 0,Y 410.825,Z 1129.959,A -85,B 0,C 180,E1 19138.53,E2 19138.53} C_VEL
LIN {X 0,Y 413.533,Z 1111.774,A -85,B 0,C 180,E1 19137.034,E2 19137.034} C_VEL
LIN {X 0,Y 415.83,Z 1094.032,A -85,B 0,C 180,E1 19135.843,E2 19135.843} C_VEL
LIN {X 0,Y 417.92,Z 1074.089,A -85,B 0,C 180,E1 19134.789,E2 19134.789} C_VEL
LIN {X 0,Y 419.526,Z 1053.852,A -85,B 0,C 180,E1 19133.994,E2 19133.994} C_VEL
LIN {X 0,Y 420.57,Z 1033.693,A -85,B 0,C 180,E1 19133.445,E2 19133.445} C_VEL
LIN {X 0,Y 427.403,Z 810.318,A -85,B 0,C 180,E1 19129.387,E2 19129.387} C_VEL
LIN {X 0,Y 420.379,Z 777.229,A -85,B 0,C 180,E1 19127.784,E2 19127.784} C_VEL
LIN {X 0,Y 421.953,Z 753.046,A -85,B 0,C 180,E1 19125.167,E2 19125.167} C_VEL
LIN {X 0,Y 416.046,Z 735.606,A -85,B 0,C 180,E1 19122.106,E2 19122.106} C_VEL
LIN {X 0,Y 415.457,Z 734.562,A -85,B 0,C 180,E1 19121.859,E2 19121.859} C_VEL
LIN {X 0,Y 421.464,Z 750.745,A -85,B 0,C 180,E1 19119.126,E2 19119.126} C_VEL
LIN {X 0,Y 417.219,Z 789.091,A -85,B 0,C 180,E1 19115.194,E2 19115.194} C_VEL
LIN {X 0,Y 412.948,Z 830.849,A -85,B 0,C 180,E1 19110.974,E2 19110.974} C_VEL
LIN {X 0,Y 410.072,Z 863.385,A -85,B 0,C 180,E1 19107.768,E2 19107.768} C_VEL
LIN {X 0,Y 411.251,Z 873.188,A -85,B 0,C 180,E1 19107.416,E2 19107.416} C_VEL
LIN {X 0,Y 404.994,Z 1034.118,A -85,B 0,C 180,E1 19103.687,E2 19103.687} C_VEL
LIN {X 0,Y 404.281,Z 1051.963,A -85,B 0,C 180,E1 19103.002,E2 19103.002} C_VEL
LIN {X 0,Y 403.242,Z 1069.309,A -85,B 0,C 180,E1 19102.065,E2 19102.065} C_VEL
LIN {X 0,Y 401.996,Z 1085.467,A -85,B 0,C 180,E1 19100.911,E2 19100.911} C_VEL
LIN {X 0,Y 400.534,Z 1101.287,A -85,B 0,C 180,E1 19099.467,E2 19099.467} C_VEL
LIN {X 0,Y 399.053,Z 1115.958,A -85,B 0,C 180,E1 19097.799,E2 19097.799} C_VEL
LIN {X 0,Y 397.705,Z 1128.404,A -85,B 0,C 180,E1 19096.055,E2 19096.055} C_VEL
LIN {X 0,Y 396.401,Z 1140.26,A -85,B 0,C 180,E1 19094.013,E2 19094.013} C_VEL
LIN {X 0,Y 395.282,Z 1150.741,A -85,B 0,C 180,E1 19091.786,E2 19091.786} C_VEL
LIN {X 0,Y 394.449,Z 1159.296,A -85,B 0,C 180,E1 19089.484,E2 19089.484} C_VEL
LIN {X 0,Y 393.869,Z 1166.446,A -85,B 0,C 180,E1 19086.983,E2 19086.983} C_VEL
LIN {X 0,Y 393.54,Z 1171.638,A -85,B 0,C 180,E1 19084.518,E2 19084.518} C_VEL
LIN {X 0,Y 393.404,Z 1175.066,A -85,B 0,C 180,E1 19082.039,E2 19082.039} C_VEL
LIN {X 0,Y 393.413,Z 1176.899,A -85,B 0,C 180,E1 19079.418,E2 19079.418} C_VEL
LIN {X 0,Y 393.574,Z 1176.97,A -85,B 0,C 180,E1 19076.766,E2 19076.766} C_VEL
LIN {X 0,Y 393.891,Z 1175.18,A -85,B 0,C 180,E1 19074.173,E2 19074.173} C_VEL
LIN {X 0,Y 394.456,Z 1171.568,A -85,B 0,C 180,E1 19071.546,E2 19071.546} C_VEL
LIN {X 0,Y 395.234,Z 1166.281,A -85,B 0,C 180,E1 19069.063,E2 19069.063} C_VEL
LIN {X 0,Y 396.373,Z 1159.011,A -85,B 0,C 180,E1 19066.581,E2 19066.581} C_VEL
LIN {X 0,Y 397.702,Z 1150.67,A -85,B 0,C 180,E1 19064.395,E2 19064.395} C_VEL
LIN {X 0,Y 399.337,Z 1140.076,A -85,B 0,C 180,E1 19062.214,E2 19062.214} C_VEL
LIN {X 0,Y 401.015,Z 1128.718,A -85,B 0,C 180,E1 19060.331,E2 19060.331} C_VEL
LIN {X 0,Y 402.755,Z 1115.529,A -85,B 0,C 180,E1 19058.585,E2 19058.585} C_VEL
LIN {X 0,Y 404.4,Z 1101.442,A -85,B 0,C 180,E1 19057.083,E2 19057.083} C_VEL
LIN {X 0,Y 405.842,Z 1085.853,A -85,B 0,C 180,E1 19055.783,E2 19055.783} C_VEL
LIN {X 0,Y 406.957,Z 1070.153,A -85,B 0,C 180,E1 19054.769,E2 19054.769} C_VEL
LIN {X 0,Y 407.743,Z 1052.132,A -85,B 0,C 180,E1 19053.935,E2 19053.935} C_VEL
LIN {X 0,Y 409.6,Z 1021.19,A -85,B 0,C 180,E1 19052.821,E2 19052.821} C_VEL
LIN {X 0,Y 417.045,Z 957.007,A -85,B 0,C 180,E1 19050.523,E2 19050.523} C_VEL
LIN {X 0,Y 423.444,Z 910.303,A -85,B 0,C 180,E1 19048.901,E2 19048.901} C_VEL
LIN {X 0,Y 433.989,Z 890.969,A -85,B 0,C 180,E1 19047.534,E2 19047.534} C_VEL
LIN {X 0,Y 435.375,Z 888.448,A -85,B 0,C 180,E1 19047.338,E2 19047.338} C_VEL
LIN {X 0,Y 443.525,Z 872.649,A -85,B 0,C 180,E1 19045.068,E2 19045.068} C_VEL
LIN {X 0,Y 448.283,Z 865.378,A -85,B 0,C 180,E1 19043.926,E2 19043.926} C_VEL
LIN {X 0,Y 444.786,Z 873.091,A -85,B 0,C 180,E1 19042.306,E2 19042.306} C_VEL
LIN {X 0,Y 443.483,Z 881.082,A -85,B 0,C 180,E1 19040.653,E2 19040.653} C_VEL
LIN {X 0,Y 444.499,Z 889.669,A -85,B 0,C 180,E1 19038.942,E2 19038.942} C_VEL
LIN {X 0,Y 447.879,Z 898.59,A -85,B 0,C 180,E1 19037.262,E2 19037.262} C_VEL
LIN {X 0,Y 453.472,Z 907.541,A -85,B 0,C 180,E1 19035.657,E2 19035.657} C_VEL
LIN {X 0,Y 461.223,Z 916.733,A -85,B 0,C 180,E1 19034.112,E2 19034.112} C_VEL
LIN {X 0,Y 450.055,Z 937.454,A -85,B 0,C 180,E1 19033.528,E2 19033.528} C_VEL
LIN {X 0,Y 440.306,Z 958.532,A -85,B 0,C 180,E1 19032.764,E2 19032.764} C_VEL
LIN {X 0,Y 431.922,Z 976.834,A -85,B 0,C 180,E1 19032.08,E2 19032.08} C_VEL
LIN {X 0,Y 426.328,Z 992.108,A -85,B 0,C 180,E1 19031.416,E2 19031.416} C_VEL
LIN {X 0,Y 421.635,Z 1022.456,A -85,B 0,C 180,E1 19031.066,E2 19031.066} C_VEL
LIN {X 0,Y 420.02,Z 1043.427,A -85,B 0,C 180,E1 19030.541,E2 19030.541} C_VEL
LIN {X 0,Y 417.419,Z 1071.84,A -85,B 0,C 180,E1 19029.574,E2 19029.574} C_VEL
LIN {X 0,Y 414.721,Z 1096.836,A -85,B 0,C 180,E1 19028.464,E2 19028.464} C_VEL
LIN {X 0,Y 411.869,Z 1122.549,A -85,B 0,C 180,E1 19027.017,E2 19027.017} C_VEL
LIN {X 0,Y 409.102,Z 1146.15,A -85,B 0,C 180,E1 19025.397,E2 19025.397} C_VEL
LIN {X 0,Y 406.369,Z 1168.708,A -85,B 0,C 180,E1 19023.531,E2 19023.531} C_VEL
LIN {X 0,Y 403.719,Z 1190.253,A -85,B 0,C 180,E1 19021.422,E2 19021.422} C_VEL
LIN {X 0,Y 401.165,Z 1210.376,A -85,B 0,C 180,E1 19019.08,E2 19019.08} C_VEL
LIN {X 0,Y 398.914,Z 1228.512,A -85,B 0,C 180,E1 19016.578,E2 19016.578} C_VEL
LIN {X 0,Y 396.951,Z 1244.718,A -85,B 0,C 180,E1 19013.925,E2 19013.925} C_VEL
LIN {X 0,Y 395.364,Z 1258.697,A -85,B 0,C 180,E1 19011.202,E2 19011.202} C_VEL
LIN {X 0,Y 394.163,Z 1270.34,A -85,B 0,C 180,E1 19008.487,E2 19008.487} C_VEL
LIN {X 0,Y 393.237,Z 1280.993,A -85,B 0,C 180,E1 19005.495,E2 19005.495} C_VEL
LIN {X 0,Y 392.692,Z 1289.512,A -85,B 0,C 180,E1 19002.5,E2 19002.5} C_VEL
LIN {X 0,Y 392.368,Z 1295.802,A -85,B 0,C 180,E1 18999.683,E2 18999.683} C_VEL
LIN {X 0,Y 392.245,Z 1300.393,A -85,B 0,C 180,E1 18996.882,E2 18996.882} C_VEL
LIN {X 0,Y 392.217,Z 1303.369,A -85,B 0,C 180,E1 18994.094,E2 18994.094} C_VEL
LIN {X 0,Y 392.205,Z 1304.889,A -85,B 0,C 180,E1 18991.169,E2 18991.169} C_VEL
LIN {X 0,Y 392.196,Z 1304.839,A -85,B 0,C 180,E1 18988.54,E2 18988.54} C_VEL
LIN {X 0,Y 392.206,Z 1303.088,A -85,B 0,C 180,E1 18985.468,E2 18985.468} C_VEL
LIN {X 0,Y 392.212,Z 1299.902,A -85,B 0,C 180,E1 18982.53,E2 18982.53} C_VEL
LIN {X 0,Y 392.362,Z 1295.094,A -85,B 0,C 180,E1 18979.577,E2 18979.577} C_VEL
LIN {X 0,Y 392.739,Z 1287.851,A -85,B 0,C 180,E1 18976.305,E2 18976.305} C_VEL
LIN {X 0,Y 393.498,Z 1278.812,A -85,B 0,C 180,E1 18973.163,E2 18973.163} C_VEL
LIN {X 0,Y 394.631,Z 1268.171,A -85,B 0,C 180,E1 18970.154,E2 18970.154} C_VEL
LIN {X 0,Y 396.178,Z 1255.959,A -85,B 0,C 180,E1 18967.287,E2 18967.287} C_VEL
LIN {X 0,Y 398.155,Z 1242.276,A -85,B 0,C 180,E1 18964.57,E2 18964.57} C_VEL
LIN {X 0,Y 400.579,Z 1226.61,A -85,B 0,C 180,E1 18961.934,E2 18961.934} C_VEL
LIN {X 0,Y 403.285,Z 1209.876,A -85,B 0,C 180,E1 18959.536,E2 18959.536} C_VEL
LIN {X 0,Y 406.271,Z 1191.66,A -85,B 0,C 180,E1 18957.318,E2 18957.318} C_VEL
LIN {X 0,Y 409.209,Z 1173.319,A -85,B 0,C 180,E1 18955.428,E2 18955.428} C_VEL
LIN {X 0,Y 412.526,Z 1152.086,A -85,B 0,C 180,E1 18953.579,E2 18953.579} C_VEL
LIN {X 0,Y 415.486,Z 1132.032,A -85,B 0,C 180,E1 18952.122,E2 18952.122} C_VEL
LIN {X 0,Y 418.569,Z 1109.236,A -85,B 0,C 180,E1 18950.782,E2 18950.782} C_VEL
LIN {X 0,Y 421.255,Z 1086.557,A -85,B 0,C 180,E1 18949.734,E2 18949.734} C_VEL
LIN {X 0,Y 423.547,Z 1063.289,A -85,B 0,C 180,E1 18948.94,E2 18948.94} C_VEL
LIN {X 0,Y 425.069,Z 1039.843,A -85,B 0,C 180,E1 18948.36,E2 18948.36} C_VEL
LIN {X 0,Y 426.347,Z 1019.788,A -85,B 0,C 180,E1 18947.986,E2 18947.986} C_VEL
LIN {X 0,Y 427.33,Z 1011.54,A -85,B 0,C 180,E1 18947.862,E2 18947.862} C_VEL
LIN {X 0,Y 438.623,Z 982.375,A -85,B 0,C 180,E1 18946.496,E2 18946.496} C_VEL
LIN {X 0,Y 447.093,Z 964.578,A -85,B 0,C 180,E1 18945.844,E2 18945.844} C_VEL
LIN {X 0,Y 459.306,Z 939.311,A -85,B 0,C 180,E1 18944.97,E2 18944.97} C_VEL
LIN {X 0,Y 468.291,Z 922.93,A -85,B 0,C 180,E1 18944.525,E2 18944.525} C_VEL
LIN {X 0,Y 458.991,Z 911.415,A -85,B 0,C 180,E1 18942.646,E2 18942.646} C_VEL
LIN {X 0,Y 452.037,Z 899.608,A -85,B 0,C 180,E1 18940.898,E2 18940.898} C_VEL
LIN {X 0,Y 446.085,Z 885.115,A -85,B 0,C 180,E1 18938.945,E2 18938.945} C_VEL
LIN {X 0,Y 442.057,Z 869.338,A -85,B 0,C 180,E1 18937.021,E2 18937.021} C_VEL
LIN {X 0,Y 439.939,Z 852.68,A -85,B 0,C 180,E1 18935.179,E2 18935.179} C_VEL
LIN {X 0,Y 439.601,Z 834.141,A -85,B 0,C 180,E1 18933.318,E2 18933.318} C_VEL
LIN {X 0,Y 441.447,Z 811.53,A -85,B 0,C 180,E1 18931.292,E2 18931.292} C_VEL
LIN {X 0,Y 445.888,Z 780.085,A -85,B 0,C 180,E1 18928.677,E2 18928.677} C_VEL
LIN {X 0,Y 436.625,Z 762.308,A -85,B 0,C 180,E1 18925.209,E2 18925.209} C_VEL
LIN {X 0,Y 428.405,Z 747.036,A -85,B 0,C 180,E1 18921.927,E2 18921.927} C_VEL
LIN {X 0,Y 421.068,Z 733.893,A -85,B 0,C 180,E1 18918.841,E2 18918.841} C_VEL
LIN {X 0,Y 414.118,Z 721.421,A -85,B 0,C 180,E1 18915.689,E2 18915.689} C_VEL
LIN {X 0,Y 407.881,Z 710.838,A -85,B 0,C 180,E1 18912.745,E2 18912.745} C_VEL
LIN {X 0,Y 404.869,Z 705.72,A -85,B 0,C 180,E1 18911.25,E2 18911.25} C_VEL
LIN {X 0,Y 402.266,Z 701.087,A -85,B 0,C 180,E1 18909.875,E2 18909.875} C_VEL
LIN {X 0,Y 399.896,Z 697.049,A -85,B 0,C 180,E1 18908.628,E2 18908.628} C_VEL
LIN {X 0,Y 398.5,Z 695.078,A -85,B 0,C 180,E1 18907.932,E2 18907.932} C_VEL
LIN {X 0,Y 396.819,Z 691.807,A -85,B 0,C 180,E1 18906.946,E2 18906.946} C_VEL
LIN {X 0,Y 396.371,Z 690.864,A -85,B 0,C 180,E1 18906.663,E2 18906.663} C_VEL
LIN {X 0,Y 394.139,Z 687.857,A -85,B 0,C 180,E1 18905.532,E2 18905.532} C_VEL
LIN {X 0,Y 393.562,Z 685.708,A -85,B 0,C 180,E1 18904.955,E2 18904.955} C_VEL
LIN {X 0,Y 393.568,Z 685.707,A -85,B 0,C 180,E1 18900.873,E2 18900.873} C_VEL
LIN {X 0,Y 393.557,Z 685.712,A -85,B 0,C 180,E1 18896.785,E2 18896.785} C_VEL
LIN {X 0,Y 393.564,Z 685.713,A -85,B 0,C 180,E1 18892.849,E2 18892.849} C_VEL
LIN {X 0,Y 393.561,Z 685.708,A -85,B 0,C 180,E1 18888.867,E2 18888.867} C_VEL
LIN {X 0,Y 393.553,Z 685.712,A -85,B 0,C 180,E1 18884.83,E2 18884.83} C_VEL
LIN {X 0,Y 393.554,Z 685.696,A -85,B 0,C 180,E1 18880.868,E2 18880.868} C_VEL
LIN {X 0,Y 393.565,Z 685.696,A -85,B 0,C 180,E1 18876.875,E2 18876.875} C_VEL
LIN {X 0,Y 393.558,Z 685.673,A -85,B 0,C 180,E1 18872.95,E2 18872.95} C_VEL
LIN {X 0,Y 393.567,Z 685.687,A -85,B 0,C 180,E1 18868.784,E2 18868.784} C_VEL
LIN {X 0,Y 393.576,Z 685.839,A -85,B 0,C 180,E1 18864.782,E2 18864.782} C_VEL
LIN {X 0,Y 394.846,Z 689.123,A -85,B 0,C 180,E1 18864.2,E2 18864.2} C_VEL
LIN {X 0,Y 396.544,Z 691.295,A -85,B 0,C 180,E1 18863.662,E2 18863.662} C_VEL
LIN {X 0,Y 398.426,Z 694.933,A -85,B 0,C 180,E1 18862.941,E2 18862.941} C_VEL
LIN {X 0,Y 399.792,Z 697.385,A -85,B 0,C 180,E1 18862.447,E2 18862.447} C_VEL
LIN {X 0,Y 404.648,Z 706.038,A -85,B 0,C 180,E1 18860.76,E2 18860.76} C_VEL
LIN {X 0,Y 411.735,Z 719.939,A -85,B 0,C 180,E1 18858.288,E2 18858.288} C_VEL
LIN {X 0,Y 419.197,Z 736.316,A -85,B 0,C 180,E1 18855.664,E2 18855.664} C_VEL
LIN {X 0,Y 425.693,Z 752.311,A -85,B 0,C 180,E1 18853.368,E2 18853.368} C_VEL
LIN {X 0,Y 424.438,Z 776.141,A -85,B 0,C 180,E1 18851.622,E2 18851.622} C_VEL
LIN {X 0,Y 427.683,Z 801.456,A -85,B 0,C 180,E1 18850.675,E2 18850.675} C_VEL
LIN {X 0,Y 420.424,Z 1036.805,A -85,B 0,C 180,E1 18846.39,E2 18846.39} C_VEL
LIN {X 0,Y 419.216,Z 1057.647,A -85,B 0,C 180,E1 18845.779,E2 18845.779} C_VEL
LIN {X 0,Y 417.489,Z 1078.174,A -85,B 0,C 180,E1 18844.916,E2 18844.916} C_VEL
LIN {X 0,Y 415.402,Z 1097.274,A -85,B 0,C 180,E1 18843.859,E2 18843.859} C_VEL
LIN {X 0,Y 413.019,Z 1115.451,A -85,B 0,C 180,E1 18842.599,E2 18842.599} C_VEL
LIN {X 0,Y 412.668,Z 1117.732,A -85,B 0,C 180,E1 18842.415,E2 18842.415} C_VEL
LIN {X 0,Y 410.832,Z 1124.585,A -85,B 0,C 180,E1 18841.937,E2 18841.937} C_VEL
LIN {X 0,Y 403.024,Z 1141.324,A -85,B 0,C 180,E1 18840.839,E2 18840.839} C_VEL
LIN {X 0,Y 401.061,Z 1147.516,A -85,B 0,C 180,E1 18840.248,E2 18840.248} C_VEL
LIN {X 0,Y 398.055,Z 1163.553,A -85,B 0,C 180,E1 18838.295,E2 18838.295} C_VEL
LIN {X 0,Y 395.148,Z 1178.458,A -85,B 0,C 180,E1 18836.121,E2 18836.121} C_VEL
LIN {X 0,Y 392.426,Z 1192.109,A -85,B 0,C 180,E1 18833.738,E2 18833.738} C_VEL
LIN {X 0,Y 389.912,Z 1204.909,A -85,B 0,C 180,E1 18831.038,E2 18831.038} C_VEL
LIN {X 0,Y 387.947,Z 1215.482,A -85,B 0,C 180,E1 18828.326,E2 18828.326} C_VEL
LIN {X 0,Y 386.485,Z 1224.177,A -85,B 0,C 180,E1 18825.607,E2 18825.607} C_VEL
LIN {X 0,Y 385.377,Z 1231.921,A -85,B 0,C 180,E1 18822.587,E2 18822.587} C_VEL
LIN {X 0,Y 384.705,Z 1237.837,A -85,B 0,C 180,E1 18819.574,E2 18819.574} C_VEL
LIN {X 0,Y 384.348,Z 1242.076,A -85,B 0,C 180,E1 18816.572,E2 18816.572} C_VEL
LIN {X 0,Y 384.192,Z 1244.678,A -85,B 0,C 180,E1 18813.58,E2 18813.58} C_VEL
LIN {X 0,Y 384.143,Z 1245.731,A -85,B 0,C 180,E1 18810.596,E2 18810.596} C_VEL
LIN {X 0,Y 384.164,Z 1245.237,A -85,B 0,C 180,E1 18807.463,E2 18807.463} C_VEL
LIN {X 0,Y 384.266,Z 1243.229,A -85,B 0,C 180,E1 18804.475,E2 18804.475} C_VEL
LIN {X 0,Y 384.54,Z 1239.675,A -85,B 0,C 180,E1 18801.476,E2 18801.476} C_VEL
LIN {X 0,Y 385.112,Z 1234.115,A -85,B 0,C 180,E1 18798.316,E2 18798.316} C_VEL
LIN {X 0,Y 386.063,Z 1226.975,A -85,B 0,C 180,E1 18795.296,E2 18795.296} C_VEL
LIN {X 0,Y 387.441,Z 1218.37,A -85,B 0,C 180,E1 18792.425,E2 18792.425} C_VEL
LIN {X 0,Y 389.31,Z 1208.024,A -85,B 0,C 180,E1 18789.624,E2 18789.624} C_VEL
LIN {X 0,Y 391.577,Z 1196.282,A -85,B 0,C 180,E1 18787.003,E2 18787.003} C_VEL
LIN {X 0,Y 394.223,Z 1183.046,A -85,B 0,C 180,E1 18784.545,E2 18784.545} C_VEL
LIN {X 0,Y 397.083,Z 1168.706,A -85,B 0,C 180,E1 18782.317,E2 18782.317} C_VEL
LIN {X 0,Y 400.116,Z 1152.874,A -85,B 0,C 180,E1 18780.261,E2 18780.261} C_VEL
LIN {X 0,Y 403.258,Z 1135.233,A -85,B 0,C 180,E1 18778.371,E2 18778.371} C_VEL
LIN {X 0,Y 406.139,Z 1117.14,A -85,B 0,C 180,E1 18776.786,E2 18776.786} C_VEL
LIN {X 0,Y 408.648,Z 1099.068,A -85,B 0,C 180,E1 18775.498,E2 18775.498} C_VEL
LIN {X 0,Y 410.913,Z 1079.493,A -85,B 0,C 180,E1 18774.388,E2 18774.388} C_VEL
LIN {X 0,Y 412.741,Z 1058.871,A -85,B 0,C 180,E1 18773.502,E2 18773.502} C_VEL
LIN {X 0,Y 414.012,Z 1038.28,A -85,B 0,C 180,E1 18772.881,E2 18772.881} C_VEL
LIN {X 0,Y 417.21,Z 938.557,A -85,B 0,C 180,E1 18771.022,E2 18771.022} C_VEL
LIN {X 0,Y 421.224,Z 811.479,A -85,B 0,C 180,E1 18768.679,E2 18768.679} C_VEL
LIN {X 0,Y 414.169,Z 777.911,A -85,B 0,C 180,E1 18767.011,E2 18767.011} C_VEL
LIN {X 0,Y 415.567,Z 756.936,A -85,B 0,C 180,E1 18764.739,E2 18764.739} C_VEL
LIN {X 0,Y 410.234,Z 741.043,A -85,B 0,C 180,E1 18761.929,E2 18761.929} C_VEL
LIN {X 0,Y 409.889,Z 740.948,A -85,B 0,C 180,E1 18761.822,E2 18761.822} C_VEL
LIN {X 0,Y 414.77,Z 754.488,A -85,B 0,C 180,E1 18759.525,E2 18759.525} C_VEL
LIN {X 0,Y 410.211,Z 793.718,A -85,B 0,C 180,E1 18755.458,E2 18755.458} C_VEL
LIN {X 0,Y 405.851,Z 835.038,A -85,B 0,C 180,E1 18751.254,E2 18751.254} C_VEL
LIN {X 0,Y 403.17,Z 864.612,A -85,B 0,C 180,E1 18748.321,E2 18748.321} C_VEL
LIN {X 0,Y 404.291,Z 874.365,A -85,B 0,C 180,E1 18747.958,E2 18747.958} C_VEL
LIN {X 0,Y 397.651,Z 1035.175,A -85,B 0,C 180,E1 18744.123,E2 18744.123} C_VEL
LIN {X 0,Y 396.893,Z 1053.148,A -85,B 0,C 180,E1 18743.416,E2 18743.416} C_VEL
LIN {X 0,Y 395.854,Z 1069.855,A -85,B 0,C 180,E1 18742.499,E2 18742.499} C_VEL
LIN {X 0,Y 394.558,Z 1086.156,A -85,B 0,C 180,E1 18741.325,E2 18741.325} C_VEL
LIN {X 0,Y 393.101,Z 1101.334,A -85,B 0,C 180,E1 18739.928,E2 18739.928} C_VEL
LIN {X 0,Y 391.603,Z 1115.599,A -85,B 0,C 180,E1 18738.304,E2 18738.304} C_VEL
LIN {X 0,Y 390.174,Z 1128.376,A -85,B 0,C 180,E1 18736.526,E2 18736.526} C_VEL
LIN {X 0,Y 388.875,Z 1139.726,A -85,B 0,C 180,E1 18734.595,E2 18734.595} C_VEL
LIN {X 0,Y 387.665,Z 1150.37,A -85,B 0,C 180,E1 18732.361,E2 18732.361} C_VEL
LIN {X 0,Y 386.725,Z 1159.465,A -85,B 0,C 180,E1 18729.976,E2 18729.976} C_VEL
LIN {X 0,Y 386.111,Z 1166.517,A -85,B 0,C 180,E1 18727.589,E2 18727.589} C_VEL
LIN {X 0,Y 385.701,Z 1172.085,A -85,B 0,C 180,E1 18725.057,E2 18725.057} C_VEL
LIN {X 0,Y 385.534,Z 1175.904,A -85,B 0,C 180,E1 18722.527,E2 18722.527} C_VEL
LIN {X 0,Y 385.519,Z 1178.08,A -85,B 0,C 180,E1 18720,E2 18720} C_VEL
LIN {X 0,Y 385.65,Z 1178.575,A -85,B 0,C 180,E1 18717.474,E2 18717.474} C_VEL
LIN {X 0,Y 385.945,Z 1177.384,A -85,B 0,C 180,E1 18714.798,E2 18714.798} C_VEL
LIN {X 0,Y 386.468,Z 1174.588,A -85,B 0,C 180,E1 18712.261,E2 18712.261} C_VEL
LIN {X 0,Y 387.23,Z 1169.862,A -85,B 0,C 180,E1 18709.666,E2 18709.666} C_VEL
LIN {X 0,Y 388.301,Z 1163.582,A -85,B 0,C 180,E1 18707.206,E2 18707.206} C_VEL
LIN {X 0,Y 389.704,Z 1155.5,A -85,B 0,C 180,E1 18704.829,E2 18704.829} C_VEL
LIN {X 0,Y 391.357,Z 1145.845,A -85,B 0,C 180,E1 18702.608,E2 18702.608} C_VEL
LIN {X 0,Y 393.041,Z 1135.477,A -85,B 0,C 180,E1 18700.689,E2 18700.689} C_VEL
LIN {X 0,Y 394.885,Z 1123.125,A -85,B 0,C 180,E1 18698.85,E2 18698.85} C_VEL
LIN {X 0,Y 396.697,Z 1109.743,A -85,B 0,C 180,E1 18697.237,E2 18697.237} C_VEL
LIN {X 0,Y 398.319,Z 1095.215,A -85,B 0,C 180,E1 18695.848,E2 18695.848} C_VEL
LIN {X 0,Y 399.711,Z 1079.743,A -85,B 0,C 180,E1 18694.676,E2 18694.676} C_VEL
LIN {X 0,Y 400.735,Z 1063.177,A -85,B 0,C 180,E1 18693.743,E2 18693.743} C_VEL
LIN {X 0,Y 402.52,Z 1032.251,A -85,B 0,C 180,E1 18692.488,E2 18692.488} C_VEL
LIN {X 0,Y 408.353,Z 984.008,A -85,B 0,C 180,E1 18690.649,E2 18690.649} C_VEL
LIN {X 0,Y 418.696,Z 914.734,A -85,B 0,C 180,E1 18688.106,E2 18688.106} C_VEL
LIN {X 0,Y 429.3,Z 896.102,A -85,B 0,C 180,E1 18686.817,E2 18686.817} C_VEL
LIN {X 0,Y 432.029,Z 891.321,A -85,B 0,C 180,E1 18686.419,E2 18686.419} C_VEL
LIN {X 0,Y 440.905,Z 876.368,A -85,B 0,C 180,E1 18684.192,E2 18684.192} C_VEL
LIN {X 0,Y 442.545,Z 874.089,A -85,B 0,C 180,E1 18683.796,E2 18683.796} C_VEL
LIN {X 0,Y 439.401,Z 881.844,A -85,B 0,C 180,E1 18682.093,E2 18682.093} C_VEL
LIN {X 0,Y 438.573,Z 889.715,A -85,B 0,C 180,E1 18680.406,E2 18680.406} C_VEL
LIN {X 0,Y 439.914,Z 897.668,A -85,B 0,C 180,E1 18678.767,E2 18678.767} C_VEL
LIN {X 0,Y 443.509,Z 906.268,A -85,B 0,C 180,E1 18677.091,E2 18677.091} C_VEL
LIN {X 0,Y 449.752,Z 915.595,A -85,B 0,C 180,E1 18675.372,E2 18675.372} C_VEL
LIN {X 0,Y 452.977,Z 919.615,A -85,B 0,C 180,E1 18674.68,E2 18674.68} C_VEL
LIN {X 0,Y 442.561,Z 939.498,A -85,B 0,C 180,E1 18674.096,E2 18674.096} C_VEL
LIN {X 0,Y 434.133,Z 957.691,A -85,B 0,C 180,E1 18673.431,E2 18673.431} C_VEL
LIN {X 0,Y 425.724,Z 975.977,A -85,B 0,C 180,E1 18672.746,E2 18672.746} C_VEL
LIN {X 0,Y 421.034,Z 988.699,A -85,B 0,C 180,E1 18672.194,E2 18672.194} C_VEL
LIN {X 0,Y 415.705,Z 1021.616,A -85,B 0,C 180,E1 18671.8,E2 18671.8} C_VEL
LIN {X 0,Y 414.028,Z 1039.789,A -85,B 0,C 180,E1 18671.332,E2 18671.332} C_VEL
LIN {X 0,Y 411.078,Z 1069.18,A -85,B 0,C 180,E1 18670.304,E2 18670.304} C_VEL
LIN {X 0,Y 408.154,Z 1094.005,A -85,B 0,C 180,E1 18669.176,E2 18669.176} C_VEL
LIN {X 0,Y 405.117,Z 1119.171,A -85,B 0,C 180,E1 18667.741,E2 18667.741} C_VEL
LIN {X 0,Y 402.121,Z 1142.986,A -85,B 0,C 180,E1 18666.09,E2 18666.09} C_VEL
LIN {X 0,Y 399.241,Z 1165.475,A -85,B 0,C 180,E1 18664.211,E2 18664.211} C_VEL
LIN {X 0,Y 396.383,Z 1187.338,A -85,B 0,C 180,E1 18662.055,E2 18662.055} C_VEL
LIN {X 0,Y 393.671,Z 1209.046,A -85,B 0,C 180,E1 18659.603,E2 18659.603} C_VEL
LIN {X 0,Y 391.654,Z 1225.166,A -85,B 0,C 180,E1 18657.439,E2 18657.439} C_VEL
LIN {X 0,Y 389.816,Z 1239.865,A -85,B 0,C 180,E1 18655.12,E2 18655.12} C_VEL
LIN {X 0,Y 388.116,Z 1253.546,A -85,B 0,C 180,E1 18652.573,E2 18652.573} C_VEL
LIN {X 0,Y 386.702,Z 1266.029,A -85,B 0,C 180,E1 18649.799,E2 18649.799} C_VEL
LIN {X 0,Y 385.67,Z 1276.378,A -85,B 0,C 180,E1 18647.036,E2 18647.036} C_VEL
LIN {X 0,Y 384.946,Z 1285.31,A -85,B 0,C 180,E1 18644.133,E2 18644.133} C_VEL
LIN {X 0,Y 384.514,Z 1292.406,A -85,B 0,C 180,E1 18641.247,E2 18641.247} C_VEL
LIN {X 0,Y 384.3,Z 1297.828,A -85,B 0,C 180,E1 18638.378,E2 18638.378} C_VEL
LIN {X 0,Y 384.239,Z 1301.54,A -85,B 0,C 180,E1 18635.526,E2 18635.526} C_VEL
LIN {X 0,Y 384.229,Z 1303.797,A -85,B 0,C 180,E1 18632.536,E2 18632.536} C_VEL
LIN {X 0,Y 384.224,Z 1304.398,A -85,B 0,C 180,E1 18629.553,E2 18629.553} C_VEL
LIN {X 0,Y 384.218,Z 1303.437,A -85,B 0,C 180,E1 18626.719,E2 18626.719} C_VEL
LIN {X 0,Y 384.228,Z 1300.87,A -85,B 0,C 180,E1 18623.876,E2 18623.876} C_VEL
LIN {X 0,Y 384.318,Z 1296.516,A -85,B 0,C 180,E1 18620.869,E2 18620.869} C_VEL
LIN {X 0,Y 384.562,Z 1290.786,A -85,B 0,C 180,E1 18617.843,E2 18617.843} C_VEL
LIN {X 0,Y 385.027,Z 1283.787,A -85,B 0,C 180,E1 18614.949,E2 18614.949} C_VEL
LIN {X 0,Y 385.97,Z 1273.997,A -85,B 0,C 180,E1 18611.733,E2 18611.733} C_VEL
LIN {X 0,Y 387.359,Z 1262.496,A -85,B 0,C 180,E1 18608.658,E2 18608.658} C_VEL
LIN {X 0,Y 389.218,Z 1249.358,A -85,B 0,C 180,E1 18605.732,E2 18605.732} C_VEL
LIN {X 0,Y 391.51,Z 1234.629,A -85,B 0,C 180,E1 18602.963,E2 18602.963} C_VEL
LIN {X 0,Y 394.054,Z 1219.184,A -85,B 0,C 180,E1 18600.495,E2 18600.495} C_VEL
LIN {X 0,Y 396.967,Z 1202.191,A -85,B 0,C 180,E1 18598.173,E2 18598.173} C_VEL
LIN {X 0,Y 400.038,Z 1184.146,A -85,B 0,C 180,E1 18596.078,E2 18596.078} C_VEL
LIN {X 0,Y 403.482,Z 1163.327,A -85,B 0,C 180,E1 18594.035,E2 18594.035} C_VEL
LIN {X 0,Y 406.809,Z 1142.856,A -85,B 0,C 180,E1 18592.356,E2 18592.356} C_VEL
LIN {X 0,Y 409.962,Z 1121.477,A -85,B 0,C 180,E1 18590.917,E2 18590.917} C_VEL
LIN {X 0,Y 413.08,Z 1098.143,A -85,B 0,C 180,E1 18589.658,E2 18589.658} C_VEL
LIN {X 0,Y 415.77,Z 1075.243,A -85,B 0,C 180,E1 18588.712,E2 18588.712} C_VEL
LIN {X 0,Y 417.926,Z 1050.88,A -85,B 0,C 180,E1 18587.984,E2 18587.984} C_VEL
LIN {X 0,Y 419.652,Z 1022.058,A -85,B 0,C 180,E1 18587.381,E2 18587.381} C_VEL
LIN {X 0,Y 420.972,Z 1010.67,A -85,B 0,C 180,E1 18587.213,E2 18587.213} C_VEL
LIN {X 0,Y 432.592,Z 981.079,A -85,B 0,C 180,E1 18585.825,E2 18585.825} C_VEL
LIN {X 0,Y 441.721,Z 962.245,A -85,B 0,C 180,E1 18585.135,E2 18585.135} C_VEL
LIN {X 0,Y 453.354,Z 938.345,A -85,B 0,C 180,E1 18584.303,E2 18584.303} C_VEL
LIN {X 0,Y 460.15,Z 925.78,A -85,B 0,C 180,E1 18583.952,E2 18583.952} C_VEL
LIN {X 0,Y 451.132,Z 913.696,A -85,B 0,C 180,E1 18582.015,E2 18582.015} C_VEL
LIN {X 0,Y 443.824,Z 899.869,A -85,B 0,C 180,E1 18580.009,E2 18580.009} C_VEL
LIN {X 0,Y 438.431,Z 884.704,A -85,B 0,C 180,E1 18578.006,E2 18578.006} C_VEL
LIN {X 0,Y 434.92,Z 867.781,A -85,B 0,C 180,E1 18575.981,E2 18575.981} C_VEL
LIN {X 0,Y 433.417,Z 849.631,A -85,B 0,C 180,E1 18574.016,E2 18574.016} C_VEL
LIN {X 0,Y 433.825,Z 830.769,A -85,B 0,C 180,E1 18572.167,E2 18572.167} C_VEL
LIN {X 0,Y 436.309,Z 807.935,A -85,B 0,C 180,E1 18570.168,E2 18570.168} C_VEL
LIN {X 0,Y 439.862,Z 784.572,A -85,B 0,C 180,E1 18568.216,E2 18568.216} C_VEL
LIN {X 0,Y 431.319,Z 767.979,A -85,B 0,C 180,E1 18564.954,E2 18564.954} C_VEL
LIN {X 0,Y 422.797,Z 752.025,A -85,B 0,C 180,E1 18561.503,E2 18561.503} C_VEL
LIN {X 0,Y 414.321,Z 736.749,A -85,B 0,C 180,E1 18557.847,E2 18557.847} C_VEL
LIN {X 0,Y 408.187,Z 726.063,A -85,B 0,C 180,E1 18555.049,E2 18555.049} C_VEL
LIN {X 0,Y 403.19,Z 717.246,A -85,B 0,C 180,E1 18552.605,E2 18552.605} C_VEL
LIN {X 0,Y 399.864,Z 711.68,A -85,B 0,C 180,E1 18550.955,E2 18550.955} C_VEL
LIN {X 0,Y 397.212,Z 707.057,A -85,B 0,C 180,E1 18549.563,E2 18549.563} C_VEL
LIN {X 0,Y 394.357,Z 702.111,A -85,B 0,C 180,E1 18548.016,E2 18548.016} C_VEL
LIN {X 0,Y 392.043,Z 698.169,A -85,B 0,C 180,E1 18546.737,E2 18546.737} C_VEL
LIN {X 0,Y 390.969,Z 696.565,A -85,B 0,C 180,E1 18546.166,E2 18546.166} C_VEL
LIN {X 0,Y 388.986,Z 693.086,A -85,B 0,C 180,E1 18545.013,E2 18545.013} C_VEL
LIN {X 0,Y 388.314,Z 691.742,A -85,B 0,C 180,E1 18544.578,E2 18544.578} C_VEL
LIN {X 0,Y 386.141,Z 688.723,A -85,B 0,C 180,E1 18543.414,E2 18543.414} C_VEL
LIN {X 0,Y 385.617,Z 686.697,A -85,B 0,C 180,E1 18542.823,E2 18542.823} C_VEL
LIN {X 0,Y 385.615,Z 686.701,A -85,B 0,C 180,E1 18538.96,E2 18538.96} C_VEL
LIN {X 0,Y 385.626,Z 686.703,A -85,B 0,C 180,E1 18534.942,E2 18534.942} C_VEL
LIN {X 0,Y 385.621,Z 686.699,A -85,B 0,C 180,E1 18530.899,E2 18530.899} C_VEL
LIN {X 0,Y 385.62,Z 686.696,A -85,B 0,C 180,E1 18526.81,E2 18526.81} C_VEL
LIN {X 0,Y 385.627,Z 686.701,A -85,B 0,C 180,E1 18522.652,E2 18522.652} C_VEL
LIN {X 0,Y 385.621,Z 686.703,A -85,B 0,C 180,E1 18518.556,E2 18518.556} C_VEL
LIN {X 0,Y 385.621,Z 686.701,A -85,B 0,C 180,E1 18514.506,E2 18514.506} C_VEL
LIN {X 0,Y 385.617,Z 686.638,A -85,B 0,C 180,E1 18510.485,E2 18510.485} C_VEL
LIN {X 0,Y 385.614,Z 686.674,A -85,B 0,C 180,E1 18506.605,E2 18506.605} C_VEL
LIN {X 0,Y 385.641,Z 686.854,A -85,B 0,C 180,E1 18506.267,E2 18506.267} C_VEL
LIN {X 0,Y 386.797,Z 689.944,A -85,B 0,C 180,E1 18505.7,E2 18505.7} C_VEL
LIN {X 0,Y 388.681,Z 692.193,A -85,B 0,C 180,E1 18505.084,E2 18505.084} C_VEL
LIN {X 0,Y 390.607,Z 696.001,A -85,B 0,C 180,E1 18504.294,E2 18504.294} C_VEL
LIN {X 0,Y 391.798,Z 697.844,A -85,B 0,C 180,E1 18503.878,E2 18503.878} C_VEL
LIN {X 0,Y 397.148,Z 707.417,A -85,B 0,C 180,E1 18501.916,E2 18501.916} C_VEL
LIN {X 0,Y 404.076,Z 720.712,A -85,B 0,C 180,E1 18499.432,E2 18499.432} C_VEL
LIN {X 0,Y 411.903,Z 737.525,A -85,B 0,C 180,E1 18496.61,E2 18496.61} C_VEL
LIN {X 0,Y 418.919,Z 754.609,A -85,B 0,C 180,E1 18494.076,E2 18494.076} C_VEL
LIN {X 0,Y 419.423,Z 756.489,A -85,B 0,C 180,E1 18493.842,E2 18493.842} C_VEL
LIN {X 0,Y 418.363,Z 776.784,A -85,B 0,C 180,E1 18492.363,E2 18492.363} C_VEL
LIN {X 0,Y 421.629,Z 802.818,A -85,B 0,C 180,E1 18491.366,E2 18491.366} C_VEL
LIN {X 0,Y 414.009,Z 1037.719,A -85,B 0,C 180,E1 18487.036,E2 18487.036} C_VEL
LIN {X 0,Y 412.748,Z 1058.453,A -85,B 0,C 180,E1 18486.418,E2 18486.418} C_VEL
LIN {X 0,Y 410.963,Z 1078.749,A -85,B 0,C 180,E1 18485.554,E2 18485.554} C_VEL
LIN {X 0,Y 408.787,Z 1097.85,A -85,B 0,C 180,E1 18484.485,E2 18484.485} C_VEL
LIN {X 0,Y 406.283,Z 1116.11,A -85,B 0,C 180,E1 18483.202,E2 18483.202} C_VEL
LIN {X 0,Y 403.38,Z 1134.365,A -85,B 0,C 180,E1 18481.617,E2 18481.617} C_VEL
LIN {X 0,Y 401.061,Z 1147.516,A -85,B 0,C 180,E1 18480.248,E2 18480.248} C_VEL
LIN {X 0,Y 399.085,Z 1153.697,A -85,B 0,C 180,E1 18479.624,E2 18479.624} C_VEL
LIN {X 0,Y 390.884,Z 1168.878,A -85,B 0,C 180,E1 18478.12,E2 18478.12} C_VEL
LIN {X 0,Y 388.87,Z 1174.355,A -85,B 0,C 180,E1 18477.382,E2 18477.382} C_VEL
LIN {X 0,Y 385.876,Z 1188.644,A -85,B 0,C 180,E1 18474.983,E2 18474.983} C_VEL
LIN {X 0,Y 383.339,Z 1200.801,A -85,B 0,C 180,E1 18472.545,E2 18472.545} C_VEL
LIN {X 0,Y 381.034,Z 1212.245,A -85,B 0,C 180,E1 18469.785,E2 18469.785} C_VEL
LIN {X 0,Y 379.166,Z 1222.275,A -85,B 0,C 180,E1 18466.817,E2 18466.817} C_VEL
LIN {X 0,Y 377.823,Z 1230.453,A -85,B 0,C 180,E1 18463.778,E2 18463.778} C_VEL
LIN {X 0,Y 376.96,Z 1236.866,A -85,B 0,C 180,E1 18460.699,E2 18460.699} C_VEL
LIN {X 0,Y 376.475,Z 1241.553,A -85,B 0,C 180,E1 18457.63,E2 18457.63} C_VEL
LIN {X 0,Y 376.248,Z 1244.749,A -85,B 0,C 180,E1 18454.419,E2 18454.419} C_VEL
LIN {X 0,Y 376.169,Z 1246.234,A -85,B 0,C 180,E1 18451.37,E2 18451.37} C_VEL
LIN {X 0,Y 376.172,Z 1246.205,A -85,B 0,C 180,E1 18448.324,E2 18448.324} C_VEL
LIN {X 0,Y 376.26,Z 1244.601,A -85,B 0,C 180,E1 18445.274,E2 18445.274} C_VEL
LIN {X 0,Y 376.483,Z 1241.476,A -85,B 0,C 180,E1 18442.215,E2 18442.215} C_VEL
LIN {X 0,Y 376.973,Z 1236.747,A -85,B 0,C 180,E1 18439.145,E2 18439.145} C_VEL
LIN {X 0,Y 377.795,Z 1230.681,A -85,B 0,C 180,E1 18436.22,E2 18436.22} C_VEL
LIN {X 0,Y 379.145,Z 1222.419,A -85,B 0,C 180,E1 18433.136,E2 18433.136} C_VEL
LIN {X 0,Y 380.971,Z 1212.569,A -85,B 0,C 180,E1 18430.21,E2 18430.21} C_VEL
LIN {X 0,Y 383.113,Z 1201.87,A -85,B 0,C 180,E1 18427.602,E2 18427.602} C_VEL
LIN {X 0,Y 385.784,Z 1189.117,A -85,B 0,C 180,E1 18425.01,E2 18425.01} C_VEL
LIN {X 0,Y 388.793,Z 1174.804,A -85,B 0,C 180,E1 18422.591,E2 18422.591} C_VEL
LIN {X 0,Y 391.911,Z 1159.651,A -85,B 0,C 180,E1 18420.456,E2 18420.456} C_VEL
LIN {X 0,Y 395.005,Z 1143.665,A -85,B 0,C 180,E1 18418.571,E2 18418.571} C_VEL
LIN {X 0,Y 398.064,Z 1126.409,A -85,B 0,C 180,E1 18416.885,E2 18416.885} C_VEL
LIN {X 0,Y 400.91,Z 1108.058,A -85,B 0,C 180,E1 18415.423,E2 18415.423} C_VEL
LIN {X 0,Y 403.281,Z 1090.198,A -85,B 0,C 180,E1 18414.276,E2 18414.276} C_VEL
LIN {X 0,Y 405.475,Z 1069.756,A -85,B 0,C 180,E1 18413.248,E2 18413.248} C_VEL
LIN {X 0,Y 407.064,Z 1049.454,A -85,B 0,C 180,E1 18412.498,E2 18412.498} C_VEL
LIN {X 0,Y 408.103,Z 1028.401,A -85,B 0,C 180,E1 18411.976,E2 18411.976} C_VEL
LIN {X 0,Y 415.319,Z 813.711,A -85,B 0,C 180,E1 18408,E2 18408} C_VEL
LIN {X 0,Y 408.031,Z 778.325,A -85,B 0,C 180,E1 18406.192,E2 18406.192} C_VEL
LIN {X 0,Y 409.257,Z 760.845,A -85,B 0,C 180,E1 18404.288,E2 18404.288} C_VEL
LIN {X 0,Y 404.845,Z 747.51,A -85,B 0,C 180,E1 18401.918,E2 18401.918} C_VEL
LIN {X 0,Y 404.319,Z 747.242,A -85,B 0,C 180,E1 18401.795,E2 18401.795} C_VEL
LIN {X 0,Y 408.147,Z 757.861,A -85,B 0,C 180,E1 18399.978,E2 18399.978} C_VEL
LIN {X 0,Y 403.314,Z 797.72,A -85,B 0,C 180,E1 18395.808,E2 18395.808} C_VEL
LIN {X 0,Y 398.884,Z 837.852,A -85,B 0,C 180,E1 18391.678,E2 18391.678} C_VEL
LIN {X 0,Y 396.246,Z 865.636,A -85,B 0,C 180,E1 18388.893,E2 18388.893} C_VEL
LIN {X 0,Y 397.353,Z 875.597,A -85,B 0,C 180,E1 18388.515,E2 18388.515} C_VEL
LIN {X 0,Y 390.308,Z 1035.857,A -85,B 0,C 180,E1 18384.575,E2 18384.575} C_VEL
LIN {X 0,Y 389.553,Z 1053.276,A -85,B 0,C 180,E1 18383.885,E2 18383.885} C_VEL
LIN {X 0,Y 388.383,Z 1071.329,A -85,B 0,C 180,E1 18382.876,E2 18382.876} C_VEL
LIN {X 0,Y 387.036,Z 1087.526,A -85,B 0,C 180,E1 18381.68,E2 18381.68} C_VEL
LIN {X 0,Y 385.448,Z 1103.374,A -85,B 0,C 180,E1 18380.182,E2 18380.182} C_VEL
LIN {X 0,Y 383.836,Z 1118.097,A -85,B 0,C 180,E1 18378.452,E2 18378.452} C_VEL
LIN {X 0,Y 382.311,Z 1131.098,A -85,B 0,C 180,E1 18376.563,E2 18376.563} C_VEL
LIN {X 0,Y 380.894,Z 1142.954,A -85,B 0,C 180,E1 18374.441,E2 18374.441} C_VEL
LIN {X 0,Y 379.693,Z 1153.299,A -85,B 0,C 180,E1 18372.162,E2 18372.162} C_VEL
LIN {X 0,Y 378.766,Z 1162.027,A -85,B 0,C 180,E1 18369.727,E2 18369.727} C_VEL
LIN {X 0,Y 378.134,Z 1169.178,A -85,B 0,C 180,E1 18367.139,E2 18367.139} C_VEL
LIN {X 0,Y 377.781,Z 1174.45,A -85,B 0,C 180,E1 18364.554,E2 18364.554} C_VEL
LIN {X 0,Y 377.635,Z 1177.9,A -85,B 0,C 180,E1 18361.973,E2 18361.973} C_VEL
LIN {X 0,Y 377.674,Z 1179.785,A -85,B 0,C 180,E1 18359.242,E2 18359.242} C_VEL
LIN {X 0,Y 377.862,Z 1179.941,A -85,B 0,C 180,E1 18356.663,E2 18356.663} C_VEL
LIN {X 0,Y 378.235,Z 1178.439,A -85,B 0,C 180,E1 18354.083,E2 18354.083} C_VEL
LIN {X 0,Y 378.898,Z 1175.056,A -85,B 0,C 180,E1 18351.349,E2 18351.349} C_VEL
LIN {X 0,Y 379.818,Z 1170.078,A -85,B 0,C 180,E1 18348.767,E2 18348.767} C_VEL
LIN {X 0,Y 381.126,Z 1163.09,A -85,B 0,C 180,E1 18346.189,E2 18346.189} C_VEL
LIN {X 0,Y 382.644,Z 1155.089,A -85,B 0,C 180,E1 18343.92,E2 18343.92} C_VEL
LIN {X 0,Y 384.37,Z 1145.698,A -85,B 0,C 180,E1 18341.811,E2 18341.811} C_VEL
LIN {X 0,Y 386.387,Z 1134.019,A -85,B 0,C 180,E1 18339.711,E2 18339.711} C_VEL
LIN {X 0,Y 388.301,Z 1122.037,A -85,B 0,C 180,E1 18337.97,E2 18337.97} C_VEL
LIN {X 0,Y 390.308,Z 1107.547,A -85,B 0,C 180,E1 18336.285,E2 18336.285} C_VEL
LIN {X 0,Y 391.9,Z 1094.021,A -85,B 0,C 180,E1 18335.024,E2 18335.024} C_VEL
LIN {X 0,Y 393.391,Z 1077.625,A -85,B 0,C 180,E1 18333.826,E2 18333.826} C_VEL
LIN {X 0,Y 394.402,Z 1061.673,A -85,B 0,C 180,E1 18332.957,E2 18332.957} C_VEL
LIN {X 0,Y 396.718,Z 1031.445,A -85,B 0,C 180,E1 18331.667,E2 18331.667} C_VEL
LIN {X 0,Y 404.856,Z 975.425,A -85,B 0,C 180,E1 18329.399,E2 18329.399} C_VEL
LIN {X 0,Y 414.288,Z 919.253,A -85,B 0,C 180,E1 18327.275,E2 18327.275} C_VEL
LIN {X 0,Y 424.758,Z 901.616,A -85,B 0,C 180,E1 18326.091,E2 18326.091} C_VEL
LIN {X 0,Y 428.554,Z 895.443,A -85,B 0,C 180,E1 18325.625,E2 18325.625} C_VEL
LIN {X 0,Y 436.98,Z 882.613,A -85,B 0,C 180,E1 18323.675,E2 18323.675} C_VEL
LIN {X 0,Y 434.243,Z 890.156,A -85,B 0,C 180,E1 18321.95,E2 18321.95} C_VEL
LIN {X 0,Y 433.76,Z 897.867,A -85,B 0,C 180,E1 18320.234,E2 18320.234} C_VEL
LIN {X 0,Y 435.377,Z 905.57,A -85,B 0,C 180,E1 18318.594,E2 18318.594} C_VEL
LIN {X 0,Y 439.177,Z 913.867,A -85,B 0,C 180,E1 18316.922,E2 18316.922} C_VEL
LIN {X 0,Y 445.068,Z 922.545,A -85,B 0,C 180,E1 18315.289,E2 18315.289} C_VEL
LIN {X 0,Y 435.094,Z 942.119,A -85,B 0,C 180,E1 18314.685,E2 18314.685} C_VEL
LIN {X 0,Y 428.425,Z 956.449,A -85,B 0,C 180,E1 18314.158,E2 18314.158} C_VEL
LIN {X 0,Y 419.949,Z 974.694,A -85,B 0,C 180,E1 18313.479,E2 18313.479} C_VEL
LIN {X 0,Y 415.988,Z 985.069,A -85,B 0,C 180,E1 18313.037,E2 18313.037} C_VEL
LIN {X 0,Y 409.813,Z 1022.479,A -85,B 0,C 180,E1 18312.551,E2 18312.551} C_VEL
LIN {X 0,Y 407.589,Z 1043.443,A -85,B 0,C 180,E1 18311.944,E2 18311.944} C_VEL
LIN {X 0,Y 404.374,Z 1070.995,A -85,B 0,C 180,E1 18310.892,E2 18310.892} C_VEL
LIN {X 0,Y 400.975,Z 1097.138,A -85,B 0,C 180,E1 18309.623,E2 18309.623} C_VEL
LIN {X 0,Y 397.691,Z 1122.059,A -85,B 0,C 180,E1 18308.101,E2 18308.101} C_VEL
LIN {X 0,Y 394.236,Z 1147.363,A -85,B 0,C 180,E1 18306.224,E2 18306.224} C_VEL
LIN {X 0,Y 389.772,Z 1182.099,A -85,B 0,C 180,E1 18303.121,E2 18303.121} C_VEL
LIN {X 0,Y 387.596,Z 1199.934,A -85,B 0,C 180,E1 18301.233,E2 18301.233} C_VEL
LIN {X 0,Y 385.313,Z 1216.808,A -85,B 0,C 180,E1 18299.115,E2 18299.115} C_VEL
LIN {X 0,Y 383.21,Z 1232.184,A -85,B 0,C 180,E1 18296.833,E2 18296.833} C_VEL
LIN {X 0,Y 381.278,Z 1246.573,A -85,B 0,C 180,E1 18294.313,E2 18294.313} C_VEL
LIN {X 0,Y 379.541,Z 1260.149,A -85,B 0,C 180,E1 18291.481,E2 18291.481} C_VEL
LIN {X 0,Y 378.239,Z 1271.418,A -85,B 0,C 180,E1 18288.655,E2 18288.655} C_VEL
LIN {X 0,Y 377.319,Z 1280.7,A -85,B 0,C 180,E1 18285.84,E2 18285.84} C_VEL
LIN {X 0,Y 376.728,Z 1288.64,A -85,B 0,C 180,E1 18282.882,E2 18282.882} C_VEL
LIN {X 0,Y 376.398,Z 1294.836,A -85,B 0,C 180,E1 18279.943,E2 18279.943} C_VEL
LIN {X 0,Y 376.267,Z 1299.379,A -85,B 0,C 180,E1 18277.022,E2 18277.022} C_VEL
LIN {X 0,Y 376.254,Z 1302.268,A -85,B 0,C 180,E1 18274.115,E2 18274.115} C_VEL
LIN {X 0,Y 376.251,Z 1303.695,A -85,B 0,C 180,E1 18271.067,E2 18271.067} C_VEL
LIN {X 0,Y 376.245,Z 1303.543,A -85,B 0,C 180,E1 18268.173,E2 18268.173} C_VEL
LIN {X 0,Y 376.241,Z 1301.763,A -85,B 0,C 180,E1 18265.243,E2 18265.243} C_VEL
LIN {X 0,Y 376.274,Z 1298.3,A -85,B 0,C 180,E1 18262.212,E2 18262.212} C_VEL
LIN {X 0,Y 376.437,Z 1293.06,A -85,B 0,C 180,E1 18259.131,E2 18259.131} C_VEL
LIN {X 0,Y 376.858,Z 1285.708,A -85,B 0,C 180,E1 18255.873,E2 18255.873} C_VEL
LIN {X 0,Y 377.657,Z 1276.64,A -85,B 0,C 180,E1 18252.593,E2 18252.593} C_VEL
LIN {X 0,Y 378.931,Z 1265.918,A -85,B 0,C 180,E1 18249.456,E2 18249.456} C_VEL
LIN {X 0,Y 380.639,Z 1253.613,A -85,B 0,C 180,E1 18246.468,E2 18246.468} C_VEL
LIN {X 0,Y 382.689,Z 1240.605,A -85,B 0,C 180,E1 18243.798,E2 18243.798} C_VEL
LIN {X 0,Y 385.36,Z 1224.931,A -85,B 0,C 180,E1 18241.06,E2 18241.06} C_VEL
LIN {X 0,Y 388.329,Z 1208.163,A -85,B 0,C 180,E1 18238.575,E2 18238.575} C_VEL
LIN {X 0,Y 391.713,Z 1189.111,A -85,B 0,C 180,E1 18236.19,E2 18236.19} C_VEL
LIN {X 0,Y 395.002,Z 1170.41,A -85,B 0,C 180,E1 18234.217,E2 18234.217} C_VEL
LIN {X 0,Y 398.414,Z 1150.298,A -85,B 0,C 180,E1 18232.424,E2 18232.424} C_VEL
LIN {X 0,Y 401.576,Z 1130.667,A -85,B 0,C 180,E1 18230.956,E2 18230.956} C_VEL
LIN {X 0,Y 404.951,Z 1107.792,A -85,B 0,C 180,E1 18229.569,E2 18229.569} C_VEL
LIN {X 0,Y 407.864,Z 1085.369,A -85,B 0,C 180,E1 18228.495,E2 18228.495} C_VEL
LIN {X 0,Y 410.405,Z 1062.142,A -85,B 0,C 180,E1 18227.67,E2 18227.67} C_VEL
LIN {X 0,Y 412.085,Z 1038.808,A -85,B 0,C 180,E1 18227.062,E2 18227.062} C_VEL
LIN {X 0,Y 413.51,Z 1019.206,A -85,B 0,C 180,E1 18226.685,E2 18226.685} C_VEL
LIN {X 0,Y 414.846,Z 1009.165,A -85,B 0,C 180,E1 18226.52,E2 18226.52} C_VEL
LIN {X 0,Y 427.042,Z 978.845,A -85,B 0,C 180,E1 18225.097,E2 18225.097} C_VEL
LIN {X 0,Y 436.136,Z 960.342,A -85,B 0,C 180,E1 18224.43,E2 18224.43} C_VEL
LIN {X 0,Y 447.498,Z 937.168,A -85,B 0,C 180,E1 18223.622,E2 18223.622} C_VEL
LIN {X 0,Y 452.152,Z 928.565,A -85,B 0,C 180,E1 18223.374,E2 18223.374} C_VEL
LIN {X 0,Y 443.356,Z 915.805,A -85,B 0,C 180,E1 18221.359,E2 18221.359} C_VEL
LIN {X 0,Y 436.608,Z 901.952,A -85,B 0,C 180,E1 18219.371,E2 18219.371} C_VEL
LIN {X 0,Y 431.62,Z 886.706,A -85,B 0,C 180,E1 18217.367,E2 18217.367} C_VEL
LIN {X 0,Y 428.39,Z 869.255,A -85,B 0,C 180,E1 18215.278,E2 18215.278} C_VEL
LIN {X 0,Y 427.191,Z 850.099,A -85,B 0,C 180,E1 18213.208,E2 18213.208} C_VEL
LIN {X 0,Y 427.947,Z 830.696,A -85,B 0,C 180,E1 18211.322,E2 18211.322} C_VEL
LIN {X 0,Y 431.003,Z 806.429,A -85,B 0,C 180,E1 18209.201,E2 18209.201} C_VEL
LIN {X 0,Y 433.712,Z 788.619,A -85,B 0,C 180,E1 18207.687,E2 18207.687} C_VEL
LIN {X 0,Y 425.339,Z 772.425,A -85,B 0,C 180,E1 18204.439,E2 18204.439} C_VEL
LIN {X 0,Y 417.199,Z 757.034,A -85,B 0,C 180,E1 18201.069,E2 18201.069} C_VEL
LIN {X 0,Y 409.31,Z 742.791,A -85,B 0,C 180,E1 18197.632,E2 18197.632} C_VEL
LIN {X 0,Y 403.207,Z 732.071,A -85,B 0,C 180,E1 18194.798,E2 18194.798} C_VEL
LIN {X 0,Y 397.854,Z 722.758,A -85,B 0,C 180,E1 18192.187,E2 18192.187} C_VEL
LIN {X 0,Y 394.857,Z 717.616,A -85,B 0,C 180,E1 18190.652,E2 18190.652} C_VEL
LIN {X 0,Y 392.167,Z 712.994,A -85,B 0,C 180,E1 18189.243,E2 18189.243} C_VEL
LIN {X 0,Y 389.288,Z 708.04,A -85,B 0,C 180,E1 18187.675,E2 18187.675} C_VEL
LIN {X 0,Y 386.486,Z 703.176,A -85,B 0,C 180,E1 18186.088,E2 18186.088} C_VEL
LIN {X 0,Y 384.22,Z 699.352,A -85,B 0,C 180,E1 18184.776,E2 18184.776} C_VEL
LIN {X 0,Y 383.491,Z 698.029,A -85,B 0,C 180,E1 18184.336,E2 18184.336} C_VEL
LIN {X 0,Y 381.182,Z 694.415,A -85,B 0,C 180,E1 18183.007,E2 18183.007} C_VEL
LIN {X 0,Y 380.619,Z 692.944,A -85,B 0,C 180,E1 18182.559,E2 18182.559} C_VEL
LIN {X 0,Y 378.389,Z 690.116,A -85,B 0,C 180,E1 18181.362,E2 18181.362} C_VEL
LIN {X 0,Y 377.692,Z 687.683,A -85,B 0,C 180,E1 18180.606,E2 18180.606} C_VEL
LIN {X 0,Y 377.681,Z 687.686,A -85,B 0,C 180,E1 18176.509,E2 18176.509} C_VEL
LIN {X 0,Y 377.675,Z 687.692,A -85,B 0,C 180,E1 18172.393,E2 18172.393} C_VEL
LIN {X 0,Y 377.678,Z 687.689,A -85,B 0,C 180,E1 18168.383,E2 18168.383} C_VEL
LIN {X 0,Y 377.689,Z 687.684,A -85,B 0,C 180,E1 18164.334,E2 18164.334} C_VEL
LIN {X 0,Y 377.681,Z 687.674,A -85,B 0,C 180,E1 18160.192,E2 18160.192} C_VEL
LIN {X 0,Y 377.681,Z 687.676,A -85,B 0,C 180,E1 18156.106,E2 18156.106} C_VEL
LIN {X 0,Y 377.686,Z 687.627,A -85,B 0,C 180,E1 18152.058,E2 18152.058} C_VEL
LIN {X 0,Y 377.688,Z 687.719,A -85,B 0,C 180,E1 18147.9,E2 18147.9} C_VEL
LIN {X 0,Y 378.928,Z 691.074,A -85,B 0,C 180,E1 18147.253,E2 18147.253} C_VEL
LIN {X 0,Y 380.919,Z 693.43,A -85,B 0,C 180,E1 18146.549,E2 18146.549} C_VEL
LIN {X 0,Y 383.036,Z 697.355,A -85,B 0,C 180,E1 18145.678,E2 18145.678} C_VEL
LIN {X 0,Y 384.186,Z 699.163,A -85,B 0,C 180,E1 18145.253,E2 18145.253} C_VEL
LIN {X 0,Y 389.554,Z 708.505,A -85,B 0,C 180,E1 18143.205,E2 18143.205} C_VEL
LIN {X 0,Y 396.666,Z 721.915,A -85,B 0,C 180,E1 18140.564,E2 18140.564} C_VEL
LIN {X 0,Y 403.929,Z 737.168,A -85,B 0,C 180,E1 18137.87,E2 18137.87} C_VEL
LIN {X 0,Y 411.249,Z 754.521,A -85,B 0,C 180,E1 18135.165,E2 18135.165} C_VEL
LIN {X 0,Y 413.28,Z 759.792,A -85,B 0,C 180,E1 18134.408,E2 18134.408} C_VEL
LIN {X 0,Y 412.355,Z 777.392,A -85,B 0,C 180,E1 18133.126,E2 18133.126} C_VEL
LIN {X 0,Y 415.643,Z 804.051,A -85,B 0,C 180,E1 18132.08,E2 18132.08} C_VEL
LIN {X 0,Y 407.655,Z 1038.434,A -85,B 0,C 180,E1 18127.707,E2 18127.707} C_VEL
LIN {X 0,Y 406.341,Z 1059.148,A -85,B 0,C 180,E1 18127.081,E2 18127.081} C_VEL
LIN {X 0,Y 404.489,Z 1079.325,A -85,B 0,C 180,E1 18126.212,E2 18126.212} C_VEL
LIN {X 0,Y 402.223,Z 1098.423,A -85,B 0,C 180,E1 18125.13,E2 18125.13} C_VEL
LIN {X 0,Y 399.597,Z 1116.76,A -85,B 0,C 180,E1 18123.827,E2 18123.827} C_VEL
LIN {X 0,Y 396.563,Z 1134.966,A -85,B 0,C 180,E1 18122.225,E2 18122.225} C_VEL
LIN {X 0,Y 393.385,Z 1152.09,A -85,B 0,C 180,E1 18120.383,E2 18120.383} C_VEL
LIN {X 0,Y 390.273,Z 1167.614,A -85,B 0,C 180,E1 18118.374,E2 18118.374} C_VEL
LIN {X 0,Y 388.87,Z 1174.355,A -85,B 0,C 180,E1 18117.382,E2 18117.382} C_VEL
LIN {X 0,Y 386.861,Z 1179.786,A -85,B 0,C 180,E1 18116.607,E2 18116.607} C_VEL
LIN {X 0,Y 378.631,Z 1193.056,A -85,B 0,C 180,E1 18114.701,E2 18114.701} C_VEL
LIN {X 0,Y 376.683,Z 1197.706,A -85,B 0,C 180,E1 18113.819,E2 18113.819} C_VEL
LIN {X 0,Y 374.175,Z 1209.237,A -85,B 0,C 180,E1 18111.145,E2 18111.145} C_VEL
LIN {X 0,Y 372.106,Z 1219.306,A -85,B 0,C 180,E1 18108.323,E2 18108.323} C_VEL
LIN {X 0,Y 370.513,Z 1227.974,A -85,B 0,C 180,E1 18105.334,E2 18105.334} C_VEL
LIN {X 0,Y 369.384,Z 1235.166,A -85,B 0,C 180,E1 18102.188,E2 18102.188} C_VEL
LIN {X 0,Y 368.7,Z 1240.513,A -85,B 0,C 180,E1 18099.049,E2 18099.049} C_VEL
LIN {X 0,Y 368.359,Z 1244.205,A -85,B 0,C 180,E1 18095.92,E2 18095.92} C_VEL
LIN {X 0,Y 368.216,Z 1246.415,A -85,B 0,C 180,E1 18092.645,E2 18092.645} C_VEL
LIN {X 0,Y 368.188,Z 1246.984,A -85,B 0,C 180,E1 18089.533,E2 18089.533} C_VEL
LIN {X 0,Y 368.243,Z 1246.066,A -85,B 0,C 180,E1 18086.419,E2 18086.419} C_VEL
LIN {X 0,Y 368.419,Z 1243.541,A -85,B 0,C 180,E1 18083.298,E2 18083.298} C_VEL
LIN {X 0,Y 368.817,Z 1239.446,A -85,B 0,C 180,E1 18080.165,E2 18080.165} C_VEL
LIN {X 0,Y 369.582,Z 1233.684,A -85,B 0,C 180,E1 18077.023,E2 18077.023} C_VEL
LIN {X 0,Y 370.757,Z 1226.543,A -85,B 0,C 180,E1 18074.033,E2 18074.033} C_VEL
LIN {X 0,Y 372.47,Z 1217.586,A -85,B 0,C 180,E1 18071.045,E2 18071.045} C_VEL
LIN {X 0,Y 374.784,Z 1206.525,A -85,B 0,C 180,E1 18068.068,E2 18068.068} C_VEL
LIN {X 0,Y 377.598,Z 1193.77,A -85,B 0,C 180,E1 18065.265,E2 18065.265} C_VEL
LIN {X 0,Y 380.617,Z 1180.192,A -85,B 0,C 180,E1 18062.8,E2 18062.8} C_VEL
LIN {X 0,Y 383.778,Z 1165.609,A -85,B 0,C 180,E1 18060.587,E2 18060.587} C_VEL
LIN {X 0,Y 387.113,Z 1149.537,A -85,B 0,C 180,E1 18058.551,E2 18058.551} C_VEL
LIN {X 0,Y 390.49,Z 1131.722,A -85,B 0,C 180,E1 18056.685,E2 18056.685} C_VEL
LIN {X 0,Y 393.574,Z 1113.601,A -85,B 0,C 180,E1 18055.137,E2 18055.137} C_VEL
LIN {X 0,Y 396.2,Z 1095.729,A -85,B 0,C 180,E1 18053.894,E2 18053.894} C_VEL
LIN {X 0,Y 398.581,Z 1075.745,A -85,B 0,C 180,E1 18052.802,E2 18052.802} C_VEL
LIN {X 0,Y 400.397,Z 1055.429,A -85,B 0,C 180,E1 18051.979,E2 18051.979} C_VEL
LIN {X 0,Y 401.569,Z 1035.275,A -85,B 0,C 180,E1 18051.413,E2 18051.413} C_VEL
LIN {X 0,Y 409.358,Z 815.32,A -85,B 0,C 180,E1 18047.272,E2 18047.272} C_VEL
LIN {X 0,Y 401.995,Z 778.789,A -85,B 0,C 180,E1 18045.345,E2 18045.345} C_VEL
LIN {X 0,Y 402.87,Z 764.41,A -85,B 0,C 180,E1 18043.762,E2 18043.762} C_VEL
LIN {X 0,Y 399.35,Z 754.039,A -85,B 0,C 180,E1 18041.855,E2 18041.855} C_VEL
LIN {X 0,Y 398.816,Z 753.78,A -85,B 0,C 180,E1 18041.731,E2 18041.731} C_VEL
LIN {X 0,Y 401.465,Z 761.497,A -85,B 0,C 180,E1 18040.407,E2 18040.407} C_VEL
LIN {X 0,Y 396.509,Z 801.024,A -85,B 0,C 180,E1 18036.243,E2 18036.243} C_VEL
LIN {X 0,Y 391.963,Z 840.666,A -85,B 0,C 180,E1 18032.123,E2 18032.123} C_VEL
LIN {X 0,Y 389.376,Z 866.73,A -85,B 0,C 180,E1 18029.482,E2 18029.482} C_VEL
LIN {X 0,Y 390.457,Z 876.807,A -85,B 0,C 180,E1 18029.093,E2 18029.093} C_VEL
LIN {X 0,Y 382.975,Z 1036.539,A -85,B 0,C 180,E1 18025.04,E2 18025.04} C_VEL
LIN {X 0,Y 382.19,Z 1054.14,A -85,B 0,C 180,E1 18024.333,E2 18024.333} C_VEL
LIN {X 0,Y 381.015,Z 1071.608,A -85,B 0,C 180,E1 18023.345,E2 18023.345} C_VEL
LIN {X 0,Y 379.615,Z 1087.994,A -85,B 0,C 180,E1 18022.126,E2 18022.126} C_VEL
LIN {X 0,Y 378.041,Z 1103.286,A -85,B 0,C 180,E1 18020.677,E2 18020.677} C_VEL
LIN {X 0,Y 376.343,Z 1118.222,A -85,B 0,C 180,E1 18018.913,E2 18018.913} C_VEL
LIN {X 0,Y 374.799,Z 1130.995,A -85,B 0,C 180,E1 18017.065,E2 18017.065} C_VEL
LIN {X 0,Y 373.389,Z 1142.353,A -85,B 0,C 180,E1 18015.055,E2 18015.055} C_VEL
LIN {X 0,Y 372.066,Z 1153.123,A -85,B 0,C 180,E1 18012.708,E2 18012.708} C_VEL
LIN {X 0,Y 371.053,Z 1162.172,A -85,B 0,C 180,E1 18010.245,E2 18010.245} C_VEL
LIN {X 0,Y 370.38,Z 1169.253,A -85,B 0,C 180,E1 18007.758,E2 18007.758} C_VEL
LIN {X 0,Y 369.939,Z 1174.872,A -85,B 0,C 180,E1 18005.117,E2 18005.117} C_VEL
LIN {X 0,Y 369.768,Z 1178.938,A -85,B 0,C 180,E1 18002.325,E2 18002.325} C_VEL
LIN {X 0,Y 369.774,Z 1181.017,A -85,B 0,C 180,E1 17999.69,E2 17999.69} C_VEL
LIN {X 0,Y 369.979,Z 1181.468,A -85,B 0,C 180,E1 17996.902,E2 17996.902} C_VEL
LIN {X 0,Y 370.364,Z 1180.281,A -85,B 0,C 180,E1 17994.268,E2 17994.268} C_VEL
LIN {X 0,Y 371.019,Z 1177.405,A -85,B 0,C 180,E1 17991.633,E2 17991.633} C_VEL
LIN {X 0,Y 372.013,Z 1172.504,A -85,B 0,C 180,E1 17988.842,E2 17988.842} C_VEL
LIN {X 0,Y 373.294,Z 1166.34,A -85,B 0,C 180,E1 17986.367,E2 17986.367} C_VEL
LIN {X 0,Y 374.966,Z 1158.228,A -85,B 0,C 180,E1 17983.9,E2 17983.9} C_VEL
LIN {X 0,Y 376.913,Z 1148.574,A -85,B 0,C 180,E1 17981.599,E2 17981.599} C_VEL
LIN {X 0,Y 379.043,Z 1137.267,A -85,B 0,C 180,E1 17979.462,E2 17979.462} C_VEL
LIN {X 0,Y 381.219,Z 1124.805,A -85,B 0,C 180,E1 17977.567,E2 17977.567} C_VEL
LIN {X 0,Y 383.245,Z 1111.487,A -85,B 0,C 180,E1 17975.942,E2 17975.942} C_VEL
LIN {X 0,Y 385.113,Z 1097.438,A -85,B 0,C 180,E1 17974.553,E2 17974.553} C_VEL
LIN {X 0,Y 386.815,Z 1080.788,A -85,B 0,C 180,E1 17973.272,E2 17973.272} C_VEL
LIN {X 0,Y 388.007,Z 1064.968,A -85,B 0,C 180,E1 17972.355,E2 17972.355} C_VEL
LIN {X 0,Y 390.561,Z 1036.39,A -85,B 0,C 180,E1 17971.032,E2 17971.032} C_VEL
LIN {X 0,Y 397.99,Z 990.218,A -85,B 0,C 180,E1 17969.033,E2 17969.033} C_VEL
LIN {X 0,Y 409.831,Z 925.478,A -85,B 0,C 180,E1 17966.477,E2 17966.477} C_VEL
LIN {X 0,Y 410.73,Z 923.111,A -85,B 0,C 180,E1 17966.362,E2 17966.362} C_VEL
LIN {X 0,Y 421.164,Z 906.334,A -85,B 0,C 180,E1 17965.266,E2 17965.266} C_VEL
LIN {X 0,Y 425.856,Z 899.027,A -85,B 0,C 180,E1 17964.72,E2 17964.72} C_VEL
LIN {X 0,Y 431.419,Z 891.294,A -85,B 0,C 180,E1 17963.485,E2 17963.485} C_VEL
LIN {X 0,Y 429.103,Z 898.811,A -85,B 0,C 180,E1 17961.698,E2 17961.698} C_VEL
LIN {X 0,Y 429.078,Z 906.301,A -85,B 0,C 180,E1 17959.973,E2 17959.973} C_VEL
LIN {X 0,Y 431.425,Z 914.761,A -85,B 0,C 180,E1 17958.129,E2 17958.129} C_VEL
LIN {X 0,Y 436.113,Z 923.346,A -85,B 0,C 180,E1 17956.363,E2 17956.363} C_VEL
LIN {X 0,Y 437.58,Z 925.446,A -85,B 0,C 180,E1 17955.951,E2 17955.951} C_VEL
LIN {X 0,Y 427.679,Z 945.345,A -85,B 0,C 180,E1 17955.294,E2 17955.294} C_VEL
LIN {X 0,Y 422.714,Z 955.809,A -85,B 0,C 180,E1 17954.915,E2 17954.915} C_VEL
LIN {X 0,Y 413.796,Z 974.897,A -85,B 0,C 180,E1 17954.196,E2 17954.196} C_VEL
LIN {X 0,Y 411.336,Z 981.366,A -85,B 0,C 180,E1 17953.935,E2 17953.935} C_VEL
LIN {X 0,Y 404.275,Z 1022.374,A -85,B 0,C 180,E1 17953.364,E2 17953.364} C_VEL
LIN {X 0,Y 401.949,Z 1041.303,A -85,B 0,C 180,E1 17952.791,E2 17952.791} C_VEL
LIN {X 0,Y 398.038,Z 1071.255,A -85,B 0,C 180,E1 17951.59,E2 17951.59} C_VEL
LIN {X 0,Y 394.539,Z 1095.667,A -85,B 0,C 180,E1 17950.354,E2 17950.354} C_VEL
LIN {X 0,Y 390.854,Z 1121.106,A -85,B 0,C 180,E1 17948.75,E2 17948.75} C_VEL
LIN {X 0,Y 387.259,Z 1145.544,A -85,B 0,C 180,E1 17946.891,E2 17946.891} C_VEL
LIN {X 0,Y 385.032,Z 1163.049,A -85,B 0,C 180,E1 17945.452,E2 17945.452} C_VEL
LIN {X 0,Y 382.853,Z 1181.492,A -85,B 0,C 180,E1 17943.799,E2 17943.799} C_VEL
LIN {X 0,Y 380.488,Z 1199.317,A -85,B 0,C 180,E1 17941.884,E2 17941.884} C_VEL
LIN {X 0,Y 377.952,Z 1216.753,A -85,B 0,C 180,E1 17939.651,E2 17939.651} C_VEL
LIN {X 0,Y 375.633,Z 1232.507,A -85,B 0,C 180,E1 17937.248,E2 17937.248} C_VEL
LIN {X 0,Y 373.566,Z 1246.739,A -85,B 0,C 180,E1 17934.68,E2 17934.68} C_VEL
LIN {X 0,Y 371.788,Z 1259.712,A -85,B 0,C 180,E1 17931.904,E2 17931.904} C_VEL
